KUKA KRL program: MyProgram_021().src

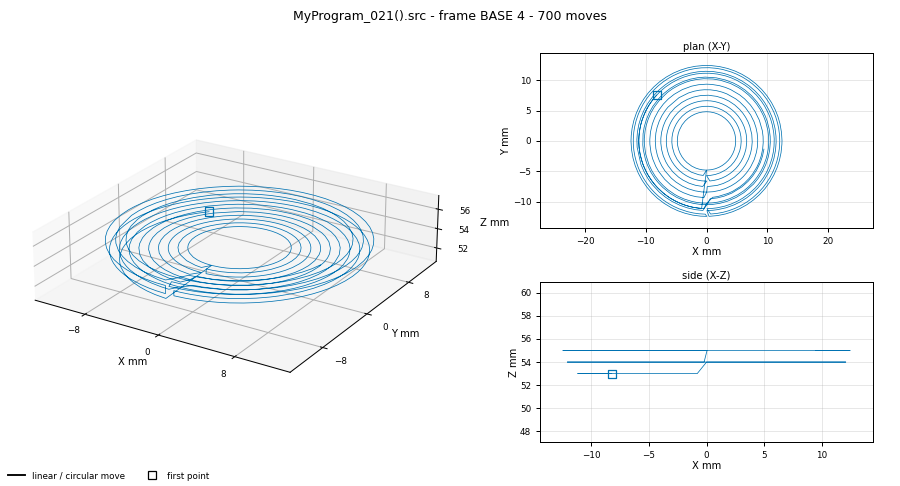
[picture p0: tool path of MyProgram_021().src in frame BASE 4, 700 of 700 moves have a stored position in this frame; points joined in program order, loops and branches not executed]
&ACCESS RVP
&REL 1
&PARAM TEMPLATE = C:\KRC\Roboter\Template\vorgabe
&PARAM EDITMASK = *
DEF MyProgram_021()
; ---- Setting reference (Base) ----
$BASE = BASE_DATA[4]

; --------------------------
; ---- Setting tool (TCP) ----
$TOOL = TOOL_DATA[3]
; --------------------------

$VEL.CP = VEL_APROX_PRINT
Startdeposition()
$VEL.CP = VEL_PRINT
LIN {X -8.217,Y 7.5391,Z 53,A 131.0651,B 24.783,C -3.3954,E1 24.879,E2 -48.9151} C_DIS
LIN {X -8.9524,Y 6.6493,Z 53,A 136.9358,B 24.785,C -3.3802,E1 24.8689,E2 -54.777} C_DIS
LIN {X -9.569,Y 5.7257,Z 53,A 142.7513,B 24.787,C -3.3647,E1 24.8603,E2 -60.5851} C_DIS
LIN {X -10.0751,Y 4.778,Z 53,A 148.3652,B 24.789,C -3.349,E1 24.8533,E2 -66.1916} C_DIS
LIN {X -10.6035,Y 3.4435,Z 53,A 154.2038,B 24.7919,C -3.3262,E1 24.8476,E2 -72.0082} C_DIS
LIN {X -10.8532,Y 2.565,Z 53,A 160.4775,B 24.7935,C -3.3127,E1 24.8431,E2 -78.2862} C_DIS
LIN {X -11.0746,Y 1.2842,Z 53,A 166.7328,B 24.7961,C -3.2919,E1 24.8405,E2 -84.5288} C_DIS
LIN {X -11.1513,Y 0.0898,Z 53,A 172.9449,B 24.7985,C -3.2728,E1 24.8398,E2 -90.7325} C_DIS
LIN {X -11.109,Y -0.9807,Z 53,A 178.5916,B 24.8006,C -3.2559,E1 24.8408,E2 -96.3727} C_DIS
LIN {X -10.9799,Y -1.9503,Z 53,A -176.0526,B 24.8024,C -3.2409,E1 24.8431,E2 -101.7244} C_DIS
LIN {X -10.6594,Y -3.2683,Z 53,A -170.537,B 24.8051,C -3.2194,E1 24.8469,E2 -107.2207} C_DIS
LIN {X -10.3597,Y -4.1289,Z 53,A -164.2287,B 24.8065,C -3.2074,E1 24.853,E2 -113.5357} C_DIS
LIN {X -9.7793,Y -5.3548,Z 53,A -158.8351,B 24.809,C -3.1872,E1 24.8596,E2 -118.9101} C_DIS
LIN {X -9.3116,Y -6.137,Z 53,A -152.506,B 24.8102,C -3.1773,E1 24.8689,E2 -125.2477} C_DIS
LIN {X -8.634,Y -7.0586,Z 53,A -146.9528,B 24.8118,C -3.1632,E1 24.8784,E2 -130.7935} C_DIS
LIN {X -7.9686,Y -7.8008,Z 53,A -141.4565,B 24.8131,C -3.1531,E1 24.889,E2 -136.2895} C_DIS
LIN {X -6.9974,Y -8.6837,Z 53,A -134.9618,B 24.8146,C -3.1401,E1 24.9027,E2 -142.7784} C_DIS
LIN {X -6.0499,Y -9.3683,Z 53,A -129.1842,B 24.8158,C -3.1301,E1 24.9159,E2 -148.5518} C_DIS
LIN {X -5.1971,Y -9.8667,Z 53,A -123.783,B 24.8165,C -3.1243,E1 24.9291,E2 -153.9546} C_DIS
LIN {X -4.1117,Y -10.3666,Z 53,A -117.7422,B 24.8172,C -3.1177,E1 24.9446,E2 -159.9938} C_DIS
LIN {X -3.1253,Y -10.7051,Z 53,A -112.1923,B 24.8176,C -3.1144,E1 24.9594,E2 -165.5458} C_DIS
LIN {X -2.0829,Y -10.9558,Z 53,A -106.4158,B 24.8178,C -3.113,E1 24.9752,E2 -171.3258} C_DIS
LIN {X -0.805,Y -11.1216,Z 53,A -100.2726,B 24.8181,C -3.1107,E1 24.9922,E2 -177.4669} C_DIS
LIN {X -0.805,Y -11.1216,Z 53,A -100.2726,B 24.8181,C -3.1107,E1 24.9922,E2 -177.4669} C_DIS
Enddeposition()
LIN {X 0.0024,Y -4.8102,Z 54,A -2.8466,B 0,C 0,E1 0.1598,E2 -269.9283} C_DIS
Startdeposition()
$VEL.CP = VEL_PRINT
LIN {X 0.8114,Y -4.7379,Z 54,A -2.8139,B 0,C 0,E1 0.1598,E2 -269.9282} C_DIS
LIN {X 1.4429,Y -4.5849,Z 54,A -2.7842,B 0,C 0,E1 0.1598,E2 -269.9282} C_DIS
LIN {X 2.0479,Y -4.3478,Z 54,A -2.7518,B 0,C 0,E1 0.1598,E2 -269.9282} C_DIS
LIN {X 2.6157,Y -4.0318,Z 54,A -2.7175,B 0,C 0,E1 0.1598,E2 -269.9281} C_DIS
LIN {X 3.1341,Y -3.6406,Z 54,A -2.6817,B 0,C 0,E1 0.1598,E2 -269.9281} C_DIS
LIN {X 3.5986,Y -3.1861,Z 54,A -2.6452,B 0,C 0,E1 0.1598,E2 -269.9281} C_DIS
LIN {X 3.9948,Y -2.6709,Z 54,A -2.6087,B 0,C 0,E1 0.1598,E2 -269.9281} C_DIS
LIN {X 4.319,Y -2.1081,Z 54,A -2.5727,B 0,C 0,E1 0.1598,E2 -269.9281} C_DIS
LIN {X 4.5648,Y -1.5065,Z 54,A -2.5379,B 0,C 0,E1 0.1598,E2 -269.9281} C_DIS
LIN {X 4.7263,Y -0.877,Z 54,A -2.5051,B 0,C 0,E1 0.1598,E2 -269.928} C_DIS
LIN {X 4.8021,Y -0.2316,Z 54,A -2.4748,B 0,C 0,E1 0.1598,E2 -269.928} C_DIS
LIN {X 4.7897,Y 0.4181,Z 54,A -2.4475,B 0,C 0,E1 0.1598,E2 -269.928} C_DIS
LIN {X 4.689,Y 1.0602,Z 54,A -2.4238,B 0,C 0,E1 0.1598,E2 -269.928} C_DIS
LIN {X 4.5023,Y 1.6826,Z 54,A -2.4041,B 0,C 0,E1 0.1598,E2 -269.9279} C_DIS
LIN {X 4.2321,Y 2.2734,Z 54,A -2.3889,B 0,C 0,E1 0.1598,E2 -269.9279} C_DIS
LIN {X 3.8894,Y 2.8255,Z 54,A -2.378,B 0,C 0,E1 0.1598,E2 -269.9278} C_DIS
LIN {X 3.4717,Y 3.3236,Z 54,A -2.3722,B 0,C 0,E1 0.1598,E2 -269.9278} C_DIS
LIN {X 2.9925,Y 3.7625,Z 54,A -2.3712,B 0,C 0,E1 0.1598,E2 -269.9278} C_DIS
LIN {X 2.4574,Y 4.1311,Z 54,A -2.3752,B 0,C 0,E1 0.1598,E2 -269.9277} C_DIS
LIN {X 1.8772,Y 4.4237,Z 54,A -2.3842,B 0,C 0,E1 0.1598,E2 -269.9277} C_DIS
LIN {X 1.263,Y 4.6358,Z 54,A -2.3978,B 0,C 0,E1 0.1598,E2 -269.9277} C_DIS
LIN {X 0.6263,Y 4.7649,Z 54,A -2.4158,B 0,C 0,E1 0.1598,E2 -269.9277} C_DIS
LIN {X -0.0221,Y 4.806,Z 54,A -2.4379,B 0,C 0,E1 0.1598,E2 -269.9277} C_DIS
LIN {X -0.6701,Y 4.7592,Z 54,A -2.4638,B 0,C 0,E1 0.1598,E2 -269.9277} C_DIS
LIN {X -1.3058,Y 4.6251,Z 54,A -2.4929,B 0,C 0,E1 0.1598,E2 -269.9277} C_DIS
LIN {X -1.9176,Y 4.4064,Z 54,A -2.5248,B 0,C 0,E1 0.1598,E2 -269.9278} C_DIS
LIN {X -2.4945,Y 4.1076,Z 54,A -2.5587,B 0,C 0,E1 0.1598,E2 -269.9278} C_DIS
LIN {X -3.0262,Y 3.734,Z 54,A -2.5941,B 0,C 0,E1 0.1598,E2 -269.928} C_DIS
LIN {X -3.5023,Y 3.2919,Z 54,A -2.6304,B 0,C 0,E1 0.1598,E2 -269.928} C_DIS
LIN {X -4.0104,Y 2.6581,Z 54,A -2.6759,B 0,C 0,E1 0.1598,E2 -269.9282} C_DIS
LIN {X -4.4662,Y 1.7787,Z 54,A -2.7298,B 0,C 0,E1 0.1598,E2 -269.9285} C_DIS
LIN {X -4.6661,Y 1.1608,Z 54,A -2.7636,B 0,C 0,E1 0.1598,E2 -269.9283} C_DIS
LIN {X -4.7799,Y 0.5214,Z 54,A -2.7949,B 0,C 0,E1 0.1598,E2 -269.9283} C_DIS
LIN {X -4.8062,Y -0.1275,Z 54,A -2.8234,B 0,C 0,E1 0.1598,E2 -269.9284} C_DIS
LIN {X -4.7448,Y -0.7741,Z 54,A -2.8486,B 0,C 0,E1 0.1598,E2 -269.9284} C_DIS
LIN {X -4.5964,Y -1.4062,Z 54,A -2.87,B 0,C 0,E1 0.1598,E2 -269.9284} C_DIS
LIN {X -4.3649,Y -2.013,Z 54,A -2.8873,B 0,C 0,E1 0.1598,E2 -269.9284} C_DIS
LIN {X -4.0539,Y -2.5829,Z 54,A -2.9001,B 0,C 0,E1 0.1598,E2 -269.9284} C_DIS
LIN {X -3.6667,Y -3.1042,Z 54,A -2.908,B 0,C 0,E1 0.1598,E2 -269.9284} C_DIS
LIN {X -3.2148,Y -3.57,Z 54,A -2.9113,B 0,C 0,E1 0.1598,E2 -269.9284} C_DIS
LIN {X -2.4084,Y -4.1653,Z 54,A -2.9069,B 0,C 0,E1 0.1598,E2 -269.9284} C_DIS
LIN {X -1.7765,Y -4.4675,Z 54,A -2.8967,B 0,C 0,E1 0.1598,E2 -269.9284} C_DIS
LIN {X -1.2443,Y -4.6427,Z 54,A -2.8847,B 0,C 0,E1 0.1598,E2 -269.9283} C_DIS
LIN {X -0.6958,Y -4.7564,Z 54,A -2.8694,B 0,C 0,E1 0.1598,E2 -269.9283} C_DIS
LIN {X 0.0024,Y -4.8102,Z 54,A -2.8461,B 0,C 0,E1 0.1598,E2 -269.9283} C_DIS
Enddeposition()
LIN {X 0.0024,Y -4.8102,Z 54,A -2.8461,B 0,C 0,E1 0.1598,E2 -269.9283} C_DIS
Startdeposition()
$VEL.CP = VEL_PRINT
LIN {X -0.5401,Y -5.685,Z 54,A -2.9028,B 0,C 0,E1 0.1598,E2 -269.9288} C_DIS
LIN {X -1.2716,Y -5.5684,Z 54,A -2.9252,B 0,C 0,E1 0.1598,E2 -269.9284} C_DIS
LIN {X -2.4971,Y -5.1425,Z 54,A -2.9519,B 0,C 0,E1 0.1598,E2 -269.9285} C_DIS
LIN {X -3.6673,Y -4.3804,Z 54,A -2.9623,B 0,C 0,E1 0.1598,E2 -269.9287} C_DIS
LIN {X -4.2148,Y -3.8632,Z 54,A -2.9605,B 0,C 0,E1 0.1598,E2 -269.9287} C_DIS
LIN {X -4.8402,Y -3.0421,Z 54,A -2.9484,B 0,C 0,E1 0.1598,E2 -269.9287} C_DIS
LIN {X -5.2993,Y -2.1427,Z 54,A -2.9267,B 0,C 0,E1 0.1598,E2 -269.9291} C_DIS
LIN {X -5.6197,Y -1.0212,Z 54,A -2.8909,B 0,C 0,E1 0.1598,E2 -269.929} C_DIS
LIN {X -5.7054,Y -0.2319,Z 54,A -2.8609,B 0,C 0,E1 0.1598,E2 -269.9286} C_DIS
LIN {X -5.6822,Y 0.5616,Z 54,A -2.8264,B 0,C 0,E1 0.1598,E2 -269.9286} C_DIS
LIN {X -5.5516,Y 1.3448,Z 54,A -2.7884,B 0,C 0,E1 0.1598,E2 -269.9285} C_DIS
LIN {X -5.3117,Y 2.1019,Z 54,A -2.7474,B 0,C 0,E1 0.1598,E2 -269.9284} C_DIS
LIN {X -4.9675,Y 2.8175,Z 54,A -2.7044,B 0,C 0,E1 0.1598,E2 -269.9284} C_DIS
LIN {X -4.5288,Y 3.4791,Z 54,A -2.6603,B 0,C 0,E1 0.1598,E2 -269.9282} C_DIS
LIN {X -4.0028,Y 4.0739,Z 54,A -2.6157,B 0,C 0,E1 0.1598,E2 -269.9281} C_DIS
LIN {X -3.3989,Y 4.5894,Z 54,A -2.5716,B 0,C 0,E1 0.1598,E2 -269.928} C_DIS
LIN {X -2.7293,Y 5.016,Z 54,A -2.5289,B 0,C 0,E1 0.1598,E2 -269.9279} C_DIS
LIN {X -2.0072,Y 5.3461,Z 54,A -2.4883,B 0,C 0,E1 0.1598,E2 -269.9278} C_DIS
LIN {X -1.2463,Y 5.5726,Z 54,A -2.4506,B 0,C 0,E1 0.1598,E2 -269.9278} C_DIS
LIN {X -0.4613,Y 5.6909,Z 54,A -2.4167,B 0,C 0,E1 0.1598,E2 -269.9277} C_DIS
LIN {X 0.3324,Y 5.7012,Z 54,A -2.387,B 0,C 0,E1 0.1598,E2 -269.9277} C_DIS
LIN {X 1.1202,Y 5.6008,Z 54,A -2.3622,B 0,C 0,E1 0.1598,E2 -269.9276} C_DIS
LIN {X 1.8858,Y 5.3907,Z 54,A -2.3429,B 0,C 0,E1 0.1598,E2 -269.9276} C_DIS
LIN {X 2.6148,Y 5.0763,Z 54,A -2.3293,B 0,C 0,E1 0.1598,E2 -269.9276} C_DIS
LIN {X 3.294,Y 4.6652,Z 54,A -2.3218,B 0,C 0,E1 0.1598,E2 -269.9276} C_DIS
LIN {X 3.9093,Y 4.1634,Z 54,A -2.3204,B 0,C 0,E1 0.1598,E2 -269.9276} C_DIS
LIN {X 4.4488,Y 3.5808,Z 54,A -2.3253,B 0,C 0,E1 0.1598,E2 -269.9277} C_DIS
LIN {X 4.9028,Y 2.9295,Z 54,A -2.3363,B 0,C 0,E1 0.1598,E2 -269.9278} C_DIS
LIN {X 5.2613,Y 2.221,Z 54,A -2.3533,B 0,C 0,E1 0.1598,E2 -269.9278} C_DIS
LIN {X 5.5168,Y 1.4694,Z 54,A -2.3759,B 0,C 0,E1 0.1598,E2 -269.9279} C_DIS
LIN {X 5.669,Y 0.6903,Z 54,A -2.4036,B 0,C 0,E1 0.1598,E2 -269.9279} C_DIS
LIN {X 5.7096,Y -0.1026,Z 54,A -2.4359,B 0,C 0,E1 0.1598,E2 -269.928} C_DIS
LIN {X 5.6414,Y -0.8937,Z 54,A -2.4722,B 0,C 0,E1 0.1598,E2 -269.928} C_DIS
LIN {X 5.4629,Y -1.6674,Z 54,A -2.5118,B 0,C 0,E1 0.1598,E2 -269.9281} C_DIS
LIN {X 5.0471,Y -2.6857,Z 54,A -2.5704,B 0,C 0,E1 0.1598,E2 -269.9284} C_DIS
LIN {X 4.5814,Y -3.4121,Z 54,A -2.6188,B 0,C 0,E1 0.1598,E2 -269.9282} C_DIS
LIN {X 4.0192,Y -4.0668,Z 54,A -2.6674,B 0,C 0,E1 0.1598,E2 -269.9282} C_DIS
LIN {X 3.1947,Y -4.7411,Z 54,A -2.7265,B 0,C 0,E1 0.1598,E2 -269.9282} C_DIS
LIN {X 2.2685,Y -5.2416,Z 54,A -2.7819,B 0,C 0,E1 0.1598,E2 -269.9282} C_DIS
LIN {X 1.4728,Y -5.517,Z 54,A -2.823,B 0,C 0,E1 0.1598,E2 -269.9282} C_DIS
LIN {X 0.6457,Y -5.6742,Z 54,A -2.86,B 0,C 0,E1 0.1598,E2 -269.9282} C_DIS
LIN {X 0.015,Y -5.7133,Z 54,A -2.8848,B 0,C 0,E1 0.1598,E2 -269.9282} C_DIS
Enddeposition()
LIN {X 0.015,Y -5.7133,Z 54,A -2.8848,B 0,C 0,E1 0.1598,E2 -269.9282} C_DIS
Startdeposition()
$VEL.CP = VEL_PRINT
LIN {X 0.5509,Y -6.5971,Z 54,A -87.2231,B 10.8099,C -0.6837,E1 10.8502,E2 -187.2658} C_DIS
LIN {X 1.2406,Y -6.5027,Z 54,A -81.5321,B 10.8098,C -0.6867,E1 10.8658,E2 -192.9584} C_DIS
LIN {X 1.9167,Y -6.338,Z 54,A -75.4134,B 10.8094,C -0.6921,E1 10.8823,E2 -199.0813} C_DIS
LIN {X 2.5716,Y -6.1025,Z 54,A -69.4109,B 10.809,C -0.699,E1 10.898,E2 -205.0878} C_DIS
LIN {X 3.1981,Y -5.7991,Z 54,A -63.3454,B 10.8084,C -0.7077,E1 10.913,E2 -211.1579} C_DIS
LIN {X 3.7889,Y -5.431,Z 54,A -57.3881,B 10.8078,C -0.7176,E1 10.9269,E2 -217.1193} C_DIS
LIN {X 4.3378,Y -5.0031,Z 54,A -51.4315,B 10.807,C -0.729,E1 10.9397,E2 -223.0801} C_DIS
LIN {X 4.8389,Y -4.52,Z 54,A -45.4727,B 10.8062,C -0.7415,E1 10.9514,E2 -229.0434} C_DIS
LIN {X 5.2864,Y -3.9869,Z 54,A -39.5211,B 10.8052,C -0.7552,E1 10.9617,E2 -234.9994} C_DIS
LIN {X 5.6755,Y -3.4099,Z 54,A -33.5711,B 10.8042,C -0.7698,E1 10.9707,E2 -240.9538} C_DIS
LIN {X 6.0017,Y -2.7951,Z 54,A -27.5272,B 10.8031,C -0.7856,E1 10.9782,E2 -247.0025} C_DIS
LIN {X 6.261,Y -2.1493,Z 54,A -21.7054,B 10.802,C -0.8012,E1 10.9838,E2 -252.8278} C_DIS
LIN {X 6.4923,Y -1.3106,Z 54,A -13.5868,B 10.8002,C -0.8245,E1 10.989,E2 -260.9553} C_DIS
LIN {X 6.6143,Y -0.3017,Z 54,A -5.704,B 10.7986,C -0.8461,E1 10.991,E2 -268.8389} C_DIS
LIN {X 6.6115,Y 0.3653,Z 54,A -0.049,B 10.7973,C -0.8621,E1 10.9906,E2 -274.497} C_DIS
LIN {X 6.5419,Y 1.0288,Z 54,A 5.6543,B 10.7961,C -0.8781,E1 10.9885,E2 -280.2032} C_DIS
LIN {X 6.4055,Y 1.6818,Z 54,A 11.4383,B 10.7948,C -0.8941,E1 10.9848,E2 -285.9903} C_DIS
LIN {X 6.2033,Y 2.3176,Z 54,A 17.1038,B 10.7935,C -0.9092,E1 10.9796,E2 -291.6578} C_DIS
LIN {X 5.9385,Y 2.9299,Z 54,A 22.7809,B 10.7923,C -0.9236,E1 10.9729,E2 -297.3367} C_DIS
LIN {X 5.6136,Y 3.5125,Z 54,A 28.5721,B 10.7911,C -0.9376,E1 10.9647,E2 -303.1298} C_DIS
LIN {X 5.2308,Y 4.0589,Z 54,A 34.0695,B 10.7901,C -0.9498,E1 10.9556,E2 -308.6272} C_DIS
LIN {X 4.7971,Y 4.5658,Z 54,A 39.8741,B 10.789,C -0.9619,E1 10.9447,E2 -314.4329} C_DIS
LIN {X 4.3134,Y 5.0254,Z 54,A 45.9575,B 10.788,C -0.9735,E1 10.9321,E2 -320.5183} C_DIS
LIN {X 3.7838,Y 5.4311,Z 54,A 51.0615,B 10.7873,C -0.9813,E1 10.9206,E2 -325.6192} C_DIS
LIN {X 3.2195,Y 5.7868,Z 54,A 57.0813,B 10.7865,C -0.99,E1 10.9062,E2 -331.6396} C_DIS
LIN {X 2.6205,Y 6.0802,Z 54,A 62.9866,B 10.7859,C -0.9968,E1 10.8912,E2 -337.5448} C_DIS
LIN {X 1.9954,Y 6.3135,Z 54,A 68.3454,B 10.7855,C -1.0012,E1 10.877,E2 -342.9003} C_DIS
LIN {X 1.3504,Y 6.4835,Z 54,A 74.382,B 10.7851,C -1.0051,E1 10.8606,E2 -348.9363} C_DIS
LIN {X 0.6911,Y 6.5857,Z 54,A 80.1461,B 10.7849,C -1.0069,E1 10.8447,E2 -354.6982} C_DIS
LIN {X 0.025,Y 6.6213,Z 54,A 86.1217,B 10.7849,C -1.0073,E1 10.828,E2 -360.6722} C_DIS
LIN {X -0.6412,Y 6.588,Z 54,A 91.4727,B 10.7851,C -1.0055,E1 10.8131,E2 -366.0184} C_DIS
LIN {X -1.3012,Y 6.4913,Z 54,A 97.5304,B 10.7853,C -1.0026,E1 10.7965,E2 -372.074} C_DIS
LIN {X -1.9473,Y 6.3258,Z 54,A 103.3049,B 10.7858,C -0.9978,E1 10.781,E2 -377.845} C_DIS
LIN {X -2.5738,Y 6.0973,Z 54,A 108.6956,B 10.7863,C -0.9917,E1 10.767,E2 -383.2303} C_DIS
LIN {X -3.1758,Y 5.8099,Z 54,A 114.887,B 10.7871,C -0.9837,E1 10.7516,E2 -389.4193} C_DIS
LIN {X -3.7448,Y 5.4616,Z 54,A 120.7148,B 10.7879,C -0.9744,E1 10.738,E2 -395.2431} C_DIS
LIN {X -4.2752,Y 5.0568,Z 54,A 126.5487,B 10.7888,C -0.9638,E1 10.7253,E2 -401.0728} C_DIS
LIN {X -4.7621,Y 4.6009,Z 54,A 132.3688,B 10.7899,C -0.952,E1 10.7137,E2 -406.8886} C_DIS
LIN {X -5.2006,Y 4.0982,Z 54,A 138.2296,B 10.791,C -0.939,E1 10.7033,E2 -412.7452} C_DIS
LIN {X -5.5864,Y 3.554,Z 54,A 144.0551,B 10.7922,C -0.9251,E1 10.6942,E2 -418.5663} C_DIS
LIN {X -5.9156,Y 2.9739,Z 54,A 149.8973,B 10.7934,C -0.9102,E1 10.6865,E2 -424.4044} C_DIS
LIN {X -6.185,Y 2.3637,Z 54,A 156.0252,B 10.7947,C -0.8942,E1 10.6801,E2 -430.5292} C_DIS
LIN {X -6.3885,Y 1.7285,Z 54,A 161.4712,B 10.796,C -0.8789,E1 10.6758,E2 -435.9697} C_DIS
LIN {X -6.5322,Y 1.0771,Z 54,A 167.4911,B 10.7973,C -0.8622,E1 10.6726,E2 -441.9864} C_DIS
LIN {X -6.6065,Y 0.4143,Z 54,A 173.2032,B 10.7986,C -0.8459,E1 10.6712,E2 -447.6943} C_DIS
LIN {X -6.6166,Y -0.2527,Z 54,A 179.2499,B 10.7999,C -0.8289,E1 10.6714,E2 -453.7385} C_DIS
LIN {X -6.5573,Y -0.9171,Z 54,A -174.9302,B 10.8011,C -0.8125,E1 10.6733,E2 -459.5552} C_DIS
LIN {X -6.4319,Y -1.5722,Z 54,A -169.0783,B 10.8023,C -0.7964,E1 10.6767,E2 -465.4045} C_DIS
LIN {X -6.2413,Y -2.2114,Z 54,A -163.2119,B 10.8034,C -0.7807,E1 10.6818,E2 -471.2685} C_DIS
LIN {X -5.9868,Y -2.828,Z 54,A -157.097,B 10.8045,C -0.7653,E1 10.6887,E2 -477.3828} C_DIS
LIN {X -5.6708,Y -3.4155,Z 54,A -151.7315,B 10.8055,C -0.7519,E1 10.6962,E2 -482.7444} C_DIS
LIN {X -5.2993,Y -3.9695,Z 54,A -145.6359,B 10.8064,C -0.7384,E1 10.706,E2 -488.8401} C_DIS
LIN {X -4.873,Y -4.4824,Z 54,A -139.8003,B 10.8072,C -0.7264,E1 10.7167,E2 -494.675} C_DIS
LIN {X -4.3971,Y -4.9498,Z 54,A -133.9626,B 10.8079,C -0.7156,E1 10.7286,E2 -500.5125} C_DIS
LIN {X -3.876,Y -5.366,Z 54,A -128.0686,B 10.8085,C -0.7061,E1 10.7417,E2 -506.407} C_DIS
LIN {X -3.3166,Y -5.7294,Z 54,A -122.302,B 10.809,C -0.6981,E1 10.7555,E2 -512.174} C_DIS
LIN {X -2.7232,Y -6.034,Z 54,A -116.6793,B 10.8094,C -0.6916,E1 10.7696,E2 -517.7967} C_DIS
LIN {X -2.1026,Y -6.2783,Z 54,A -110.7462,B 10.8098,C -0.6866,E1 10.7852,E2 -523.7319} C_DIS
LIN {X -1.4603,Y -6.4582,Z 54,A -104.7879,B 10.81,C -0.6834,E1 10.8013,E2 -529.6929} C_DIS
LIN {X -0.8028,Y -6.5706,Z 54,A -99.091,B 10.81,C -0.6817,E1 10.8171,E2 -535.3916} C_DIS
LIN {X 0.0293,Y -6.6199,Z 54,A -94.6585,B 10.8102,C -0.679,E1 10.8294,E2 -539.8122} C_DIS
Enddeposition()
LIN {X 0.0293,Y -6.6199,Z 54,A -94.6585,B 10.8102,C -0.679,E1 10.8294,E2 -539.8122} C_DIS
Startdeposition()
$VEL.CP = VEL_PRINT
LIN {X -0.6225,Y -7.5046,Z 54,A -102.6208,B 16.025,C -1.3921,E1 16.0632,E2 -532.9802} C_DIS
LIN {X -1.8167,Y -7.3038,Z 54,A -109.992,B 16.0245,C -1.398,E1 16.0431,E2 -525.6172} C_DIS
LIN {X -2.8776,Y -6.9579,Z 54,A -119.7083,B 16.0239,C -1.4043,E1 16.0175,E2 -515.8927} C_DIS
LIN {X -3.8717,Y -6.4538,Z 54,A -127.4228,B 16.023,C -1.4152,E1 15.9986,E2 -508.1826} C_DIS
LIN {X -4.5958,Y -5.9636,Z 54,A -134.6216,B 16.0221,C -1.4258,E1 15.9823,E2 -500.9818} C_DIS
LIN {X -5.5747,Y -5.0632,Z 54,A -145.3901,B 16.0203,C -1.4458,E1 15.961,E2 -490.213} C_DIS
LIN {X -6.3278,Y -4.0739,Z 54,A -152.413,B 16.0186,C -1.4655,E1 15.9494,E2 -483.207} C_DIS
LIN {X -6.6994,Y -3.4399,Z 54,A -160.3978,B 16.0171,C -1.4816,E1 15.9386,E2 -475.2132} C_DIS
LIN {X -7.1179,Y -2.4589,Z 54,A -168.4783,B 16.0152,C -1.5033,E1 15.9306,E2 -467.1385} C_DIS
LIN {X -7.3822,Y -1.4676,Z 54,A -175.4984,B 16.0132,C -1.5243,E1 15.926,E2 -460.1283} C_DIS
LIN {X -7.5214,Y -0.3734,Z 54,A 175.9813,B 16.011,C -1.5487,E1 15.9236,E2 -451.6145} C_DIS
LIN {X -7.5155,Y 0.4617,Z 54,A 169.1679,B 16.0091,C -1.5679,E1 15.9242,E2 -444.8049} C_DIS
LIN {X -7.3994,Y 1.4007,Z 54,A 161.3843,B 16.0071,C -1.5896,E1 15.9276,E2 -437.0258} C_DIS
LIN {X -7.113,Y 2.459,Z 54,A 153.6683,B 16.0048,C -1.6125,E1 15.9337,E2 -429.3211} C_DIS
LIN {X -6.7458,Y 3.3445,Z 54,A 146.0273,B 16.0028,C -1.6326,E1 15.9425,E2 -421.686} C_DIS
LIN {X -6.0298,Y 4.5097,Z 54,A 134.9592,B 16.0002,C -1.6592,E1 15.9595,E2 -410.6256} C_DIS
LIN {X -5.1947,Y 5.4498,Z 54,A 124.8201,B 15.998,C -1.6805,E1 15.9792,E2 -400.4935} C_DIS
LIN {X -4.0818,Y 6.3282,Z 54,A 114.6963,B 15.996,C -1.6996,E1 16.002,E2 -390.3826} C_DIS
LIN {X -3.1479,Y 6.8357,Z 54,A 106.9875,B 15.9948,C -1.7112,E1 16.0212,E2 -382.6825} C_DIS
LIN {X -2.1551,Y 7.2149,Z 54,A 98.4866,B 15.994,C -1.7194,E1 16.0436,E2 -374.1855} C_DIS
LIN {X -1.0372,Y 7.4539,Z 54,A 90.2017,B 15.9934,C -1.7254,E1 16.0663,E2 -365.9084} C_DIS
LIN {X 0.2973,Y 7.5246,Z 54,A 78.7875,B 15.9934,C -1.7252,E1 16.0981,E2 -354.4929} C_DIS
LIN {X 1.6715,Y 7.3371,Z 54,A 69.3006,B 15.9936,C -1.7231,E1 16.1242,E2 -345.015} C_DIS
LIN {X 2.8177,Y 6.9834,Z 54,A 60.6987,B 15.9943,C -1.7167,E1 16.1469,E2 -336.4172} C_DIS
LIN {X 3.6825,Y 6.5674,Z 54,A 52.9985,B 15.9953,C -1.7066,E1 16.166,E2 -328.7149} C_DIS
LIN {X 4.6404,Y 5.9293,Z 54,A 43.8028,B 15.9969,C -1.6913,E1 16.1869,E2 -319.5156} C_DIS
LIN {X 5.4921,Y 5.1453,Z 54,A 35.6502,B 15.9984,C -1.6764,E1 16.2033,E2 -311.3644} C_DIS
LIN {X 5.9993,Y 4.543,Z 54,A 29.3624,B 15.9999,C -1.662,E1 16.2142,E2 -305.0724} C_DIS
LIN {X 6.4398,Y 3.8903,Z 54,A 23.8542,B 16.0011,C -1.6496,E1 16.2225,E2 -299.5641} C_DIS
LIN {X 6.813,Y 3.197,Z 54,A 17.6229,B 16.0028,C -1.6333,E1 16.2303,E2 -293.3276} C_DIS
LIN {X 7.1086,Y 2.4672,Z 54,A 11.9864,B 16.0042,C -1.6187,E1 16.2359,E2 -287.6893} C_DIS
LIN {X 7.451,Y 1.0886,Z 54,A -0.0547,B 16.0077,C -1.5827,E1 16.2427,E2 -275.6318} C_DIS
LIN {X 7.5274,Y -0.1798,Z 54,A -8.7198,B 16.01,C -1.5589,E1 16.2433,E2 -266.9643} C_DIS
LIN {X 7.4365,Y -1.1791,Z 54,A -16.2028,B 16.012,C -1.5373,E1 16.2408,E2 -259.4749} C_DIS
LIN {X 7.233,Y -2.097,Z 54,A -23.6408,B 16.0141,C -1.5155,E1 16.2356,E2 -252.0278} C_DIS
LIN {X 6.8961,Y -3.023,Z 54,A -31.0943,B 16.0159,C -1.495,E1 16.2279,E2 -244.5669} C_DIS
LIN {X 6.4181,Y -3.9328,Z 54,A -38.3227,B 16.0176,C -1.477,E1 16.218,E2 -237.3344} C_DIS
LIN {X 5.9631,Y -4.5964,Z 54,A -44.8089,B 16.019,C -1.4605,E1 16.2073,E2 -230.8395} C_DIS
LIN {X 5.4213,Y -5.2248,Z 54,A -51.1979,B 16.0203,C -1.446,E1 16.1952,E2 -224.4438} C_DIS
LIN {X 4.5718,Y -5.9821,Z 54,A -59.6646,B 16.0218,C -1.4295,E1 16.177,E2 -215.97} C_DIS
LIN {X 3.6739,Y -6.5678,Z 54,A -67.1039,B 16.0227,C -1.4182,E1 16.1593,E2 -208.5282} C_DIS
LIN {X 2.7544,Y -7.0092,Z 54,A -76.2961,B 16.024,C -1.4039,E1 16.1358,E2 -199.3206} C_DIS
LIN {X 1.7894,Y -7.3144,Z 54,A -84.2551,B 16.0246,C -1.3964,E1 16.1143,E2 -191.3546} C_DIS
LIN {X 0.1158,Y -7.5288,Z 54,A -95.2263,B 16.0248,C -1.3945,E1 16.0838,E2 -180.3877} C_DIS
LIN {X 0.1158,Y -7.5288,Z 54,A -95.2263,B 16.0248,C -1.3945,E1 16.0838,E2 -180.3877} C_DIS
Enddeposition()
LIN {X 0.0276,Y -8.431,Z 54,A -95.6356,B 21.2021,C -2.3401,E1 21.3276,E2 -181.2403} C_DIS
Startdeposition()
$VEL.CP = VEL_PRINT
LIN {X 1.1282,Y -8.3607,Z 54,A -86.6538,B 21.2013,C -2.3478,E1 21.3526,E2 -190.237} C_DIS
LIN {X 2.1816,Y -8.1461,Z 54,A -80.552,B 21.201,C -2.3503,E1 21.3692,E2 -196.3356} C_DIS
LIN {X 3.1517,Y -7.8259,Z 54,A -72.727,B 21.1998,C -2.3618,E1 21.3897,E2 -204.1731} C_DIS
LIN {X 4.0868,Y -7.3743,Z 54,A -66.1117,B 21.1988,C -2.3711,E1 21.4062,E2 -210.7922} C_DIS
LIN {X 4.793,Y -6.9366,Z 54,A -60.5207,B 21.1977,C -2.3811,E1 21.4192,E2 -216.3889} C_DIS
LIN {X 5.4529,Y -6.4319,Z 54,A -55.0288,B 21.1965,C -2.392,E1 21.4312,E2 -221.8859} C_DIS
LIN {X 6.0604,Y -5.865,Z 54,A -49.224,B 21.1951,C -2.4054,E1 21.4428,E2 -227.6986} C_DIS
LIN {X 6.6073,Y -5.2395,Z 54,A -43.6532,B 21.1936,C -2.4189,E1 21.4527,E2 -233.2759} C_DIS
LIN {X 7.2505,Y -4.3132,Z 54,A -35.7516,B 21.1913,C -2.4402,E1 21.4647,E2 -241.189} C_DIS
LIN {X 7.8487,Y -3.0961,Z 54,A -26.2647,B 21.1883,C -2.4677,E1 21.4756,E2 -250.6899} C_DIS
LIN {X 8.2114,Y -1.9171,Z 54,A -18.4973,B 21.1858,C -2.4893,E1 21.4814,E2 -258.4634} C_DIS
LIN {X 8.3703,Y -1.0261,Z 54,A -12.4611,B 21.1838,C -2.5072,E1 21.4839,E2 -264.5064} C_DIS
LIN {X 8.434,Y 0.1704,Z 54,A -4.3489,B 21.1811,C -2.5315,E1 21.4845,E2 -272.6281} C_DIS
LIN {X 8.3439,Y 1.2438,Z 54,A 3.097,B 21.1785,C -2.554,E1 21.4822,E2 -280.0833} C_DIS
LIN {X 8.1431,Y 2.2032,Z 54,A 9.6166,B 21.1763,C -2.5726,E1 21.478,E2 -286.6089} C_DIS
LIN {X 7.8382,Y 3.1191,Z 54,A 16.8641,B 21.1738,C -2.5943,E1 21.4709,E2 -293.8678} C_DIS
LIN {X 7.284,Y 4.2492,Z 54,A 24.373,B 21.1718,C -2.6112,E1 21.4611,E2 -301.3762} C_DIS
LIN {X 6.4171,Y 5.4748,Z 54,A 35.8226,B 21.1684,C -2.6404,E1 21.4417,E2 -312.8412} C_DIS
LIN {X 5.4929,Y 6.3959,Z 54,A 43.1332,B 21.1671,C -2.651,E1 21.4269,E2 -320.1452} C_DIS
LIN {X 4.8107,Y 6.929,Z 54,A 50.8409,B 21.1651,C -2.6678,E1 21.4094,E2 -327.867} C_DIS
LIN {X 3.3598,Y 7.7376,Z 54,A 60.6789,B 21.1641,C -2.6763,E1 21.3849,E2 -337.6964} C_DIS
LIN {X 2.5856,Y 8.0297,Z 54,A 66.6613,B 21.1634,C -2.6821,E1 21.3691,E2 -343.6807} C_DIS
LIN {X 1.6802,Y 8.2667,Z 54,A 72.7242,B 21.1631,C -2.6846,E1 21.3526,E2 -349.7404} C_DIS
LIN {X 0.6449,Y 8.4114,Z 54,A 79.6912,B 21.163,C -2.6855,E1 21.3333,E2 -356.7041} C_DIS
LIN {X -0.3753,Y 8.4245,Z 54,A 86.5907,B 21.1631,C -2.6842,E1 21.3141,E2 -363.6} C_DIS
LIN {X -1.1879,Y 8.3476,Z 54,A 92.1541,B 21.1635,C -2.6814,E1 21.2986,E2 -369.1601} C_DIS
LIN {X -1.9893,Y 8.1933,Z 54,A 97.5698,B 21.164,C -2.6768,E1 21.2839,E2 -374.571} C_DIS
LIN {X -2.9656,Y 7.8971,Z 54,A 106.1126,B 21.1647,C -2.6708,E1 21.2614,E2 -383.1169} C_DIS
LIN {X -4.5341,Y 7.114,Z 54,A 119.2976,B 21.167,C -2.6522,E1 21.2296,E2 -396.2969} C_DIS
LIN {X -6.3433,Y 5.561,Z 54,A 132.236,B 21.1712,C -2.6163,E1 21.2033,E2 -409.1985} C_DIS
LIN {X -6.797,Y 4.9972,Z 54,A 138.1223,B 21.1727,C -2.6039,E1 21.1933,E2 -415.0838} C_DIS
LIN {X -7.3259,Y 4.1838,Z 54,A 145.1701,B 21.1748,C -2.5862,E1 21.1831,E2 -422.1255} C_DIS
LIN {X -7.7974,Y 3.2156,Z 54,A 151.5342,B 21.1771,C -2.5661,E1 21.1758,E2 -428.4753} C_DIS
LIN {X -8.1419,Y 2.2076,Z 54,A 159.4933,B 21.1796,C -2.5445,E1 21.1691,E2 -436.4289} C_DIS
LIN {X -8.3386,Y 1.2767,Z 54,A 166.1394,B 21.1818,C -2.5251,E1 21.1658,E2 -443.0678} C_DIS
LIN {X -8.437,Y 0.0383,Z 54,A 175.2854,B 21.1847,C -2.4991,E1 21.1648,E2 -452.2073} C_DIS
LIN {X -8.3426,Y -1.2521,Z 54,A -176.4078,B 21.1876,C -2.4733,E1 21.1673,E2 -460.5015} C_DIS
LIN {X -8.087,Y -2.4023,Z 54,A -168.478,B 21.1902,C -2.4503,E1 21.1728,E2 -468.4226} C_DIS
LIN {X -7.7669,Y -3.2808,Z 54,A -162.6573,B 21.1921,C -2.4332,E1 21.1787,E2 -474.2346} C_DIS
LIN {X -7.3595,Y -4.1226,Z 54,A -155.721,B 21.1939,C -2.4165,E1 21.1876,E2 -481.1688} C_DIS
LIN {X -6.848,Y -4.9279,Z 54,A -148.0345,B 21.1956,C -2.4012,E1 21.1999,E2 -488.8579} C_DIS
LIN {X -5.7863,Y -6.1377,Z 54,A -138.2423,B 21.198,C -2.3783,E1 21.2186,E2 -498.6373} C_DIS
LIN {X -5.0175,Y -6.7826,Z 54,A -131.5962,B 21.1993,C -2.3664,E1 21.2332,E2 -505.2798} C_DIS
LIN {X -3.9696,Y -7.4436,Z 54,A -121.7245,B 21.2003,C -2.3566,E1 21.257,E2 -515.1595} C_DIS
LIN {X -3.0466,Y -7.8673,Z 54,A -115.5849,B 21.2011,C -2.3489,E1 21.2729,E2 -521.2941} C_DIS
LIN {X -1.8873,Y -8.2177,Z 54,A -108.0527,B 21.2018,C -2.3428,E1 21.2931,E2 -528.823} C_DIS
LIN {X -0.8347,Y -8.3951,Z 54,A -100.2493,B 21.2018,C -2.3424,E1 21.3147,E2 -536.6324} C_DIS
LIN {X 0.0276,Y -8.431,Z 54,A -96.3606,B 21.2023,C -2.3382,E1 21.3255,E2 -540.5102} C_DIS
Enddeposition()
LIN {X 0.0276,Y -8.431,Z 54,A -96.3606,B 21.2023,C -2.3382,E1 21.3255,E2 -540.5102} C_DIS
Startdeposition()
$VEL.CP = VEL_PRINT
LIN {X -0.4267,Y -9.3338,Z 54,A -101.7866,B 24.8148,C -3.1386,E1 24.9882,E2 -536.0191} C_DIS
LIN {X -1.7131,Y -9.1852,Z 54,A -109.633,B 24.8145,C -3.1406,E1 24.9665,E2 -528.1711} C_DIS
LIN {X -2.6403,Y -8.9621,Z 54,A -115.8561,B 24.8142,C -3.1433,E1 24.9498,E2 -521.9447} C_DIS
LIN {X -3.7967,Y -8.5324,Z 54,A -121.3225,B 24.8129,C -3.1546,E1 24.9356,E2 -516.4936} C_DIS
LIN {X -4.5899,Y -8.1367,Z 54,A -129.6831,B 24.8127,C -3.1564,E1 24.9149,E2 -508.1141} C_DIS
LIN {X -5.8923,Y -7.2514,Z 54,A -138.7667,B 24.8106,C -3.1732,E1 24.8946,E2 -499.0384} C_DIS
LIN {X -6.8805,Y -6.3198,Z 54,A -147.8405,B 24.8086,C -3.1898,E1 24.8769,E2 -489.9655} C_DIS
LIN {X -7.856,Y -5.0569,Z 54,A -155.6466,B 24.8057,C -3.2142,E1 24.8642,E2 -482.1798} C_DIS
LIN {X -8.3477,Y -4.1947,Z 54,A -163.2323,B 24.8038,C -3.2298,E1 24.8542,E2 -474.5912} C_DIS
LIN {X -8.8563,Y -2.9775,Z 54,A -170.2475,B 24.801,C -3.2526,E1 24.8472,E2 -467.5914} C_DIS
LIN {X -9.1423,Y -1.92,Z 54,A -178.3476,B 24.7985,C -3.2726,E1 24.842,E2 -459.4918} C_DIS
LIN {X -9.3241,Y -0.5379,Z 54,A 174.2677,B 24.7953,C -3.2987,E1 24.8399,E2 -452.1252} C_DIS
LIN {X -9.3366,Y 0.2473,Z 54,A 169.4988,B 24.7934,C -3.3136,E1 24.8399,E2 -447.3634} C_DIS
LIN {X -9.224,Y 1.4786,Z 54,A 161.5798,B 24.7905,C -3.3371,E1 24.8425,E2 -439.4534} C_DIS
LIN {X -8.9122,Y 2.7996,Z 54,A 153.0447,B 24.7873,C -3.3625,E1 24.8485,E2 -430.9295} C_DIS
LIN {X -8.5158,Y 3.8321,Z 54,A 146.6818,B 24.7847,C -3.3825,E1 24.8552,E2 -424.5792} C_DIS
LIN {X -7.8959,Y 4.9926,Z 54,A 137.6553,B 24.7818,C -3.4048,E1 24.8677,E2 -415.559} C_DIS
LIN {X -7.1061,Y 6.0634,Z 54,A 129.4411,B 24.7792,C -3.4255,E1 24.8819,E2 -407.356} C_DIS
LIN {X -6.2611,Y 6.9355,Z 54,A 122.1458,B 24.7769,C -3.4426,E1 24.8965,E2 -400.0714} C_DIS
LIN {X -5.3216,Y 7.6774,Z 54,A 114.7177,B 24.775,C -3.4573,E1 24.9131,E2 -392.652} C_DIS
LIN {X -3.968,Y 8.4577,Z 54,A 103.426,B 24.7733,C -3.4704,E1 24.9411,E2 -381.3609} C_DIS
LIN {X -2.4474,Y 9.0159,Z 54,A 94.7461,B 24.7716,C -3.4836,E1 24.9641,E2 -372.6972} C_DIS
LIN {X -1.3109,Y 9.2509,Z 54,A 87.9433,B 24.7708,C -3.4893,E1 24.9828,E2 -365.9015} C_DIS
LIN {X -0.0062,Y 9.3434,Z 54,A 80.5908,B 24.7702,C -3.4936,E1 25.0033,E2 -358.5577} C_DIS
LIN {X 0.8706,Y 9.3027,Z 54,A 74.0291,B 24.7707,C -3.4899,E1 25.0216,E2 -351.9905} C_DIS
LIN {X 2.1604,Y 9.0902,Z 54,A 65.9239,B 24.7712,C -3.4861,E1 25.0437,E2 -343.8863} C_DIS
LIN {X 3.11,Y 8.8095,Z 54,A 60.4635,B 24.7716,C -3.4835,E1 25.0582,E2 -338.4303} C_DIS
LIN {X 3.975,Y 8.4544,Z 54,A 54.4012,B 24.7726,C -3.4759,E1 25.0736,E2 -332.3651} C_DIS
LIN {X 5.4357,Y 7.5985,Z 54,A 44.6319,B 24.7742,C -3.4632,E1 25.0967,E2 -322.5969} C_DIS
LIN {X 6.2787,Y 6.9194,Z 54,A 38.3466,B 24.7756,C -3.4526,E1 25.11,E2 -316.3107} C_DIS
LIN {X 7.2298,Y 5.9185,Z 54,A 27.7525,B 24.7795,C -3.4232,E1 25.1296,E2 -305.6943} C_DIS
LIN {X 7.9841,Y 4.8499,Z 54,A 20.4375,B 24.7816,C -3.4069,E1 25.1404,E2 -298.3775} C_DIS
LIN {X 8.7007,Y 3.4055,Z 54,A 10.8679,B 24.7848,C -3.3814,E1 25.1512,E2 -288.7996} C_DIS
LIN {X 9.1891,Y 1.6903,Z 54,A 1.1359,B 24.7881,C -3.3562,E1 25.1578,E2 -279.064} C_DIS
LIN {X 9.3145,Y 0.721,Z 54,A -5.041,B 24.7905,C -3.3368,E1 25.1596,E2 -272.8776} C_DIS
LIN {X 9.3381,Y -0.2783,Z 54,A -10.969,B 24.7928,C -3.319,E1 25.1596,E2 -266.9427} C_DIS
LIN {X 9.2407,Y -1.3751,Z 54,A -17.9721,B 24.7956,C -3.2965,E1 25.1573,E2 -259.9277} C_DIS
LIN {X 9.001,Y -2.4896,Z 54,A -24.3489,B 24.7978,C -3.2789,E1 25.1532,E2 -253.5459} C_DIS
LIN {X 8.6252,Y -3.5881,Z 54,A -30.8524,B 24.7999,C -3.2612,E1 25.147,E2 -247.037} C_DIS
LIN {X 8.2762,Y -4.3361,Z 54,A -37.3776,B 24.8028,C -3.2381,E1 25.1389,E2 -240.4918} C_DIS
LIN {X 7.5866,Y -5.4456,Z 54,A -43.2856,B 24.804,C -3.2283,E1 25.13,E2 -234.5903} C_DIS
LIN {X 7.0283,Y -6.1543,Z 54,A -50.4094,B 24.8068,C -3.2054,E1 25.1174,E2 -227.445} C_DIS
LIN {X 6.2437,Y -6.9511,Z 54,A -57.1307,B 24.8086,C -3.1902,E1 25.1039,E2 -220.7156} C_DIS
LIN {X 5.5183,Y -7.54,Z 54,A -63.0226,B 24.8101,C -3.1776,E1 25.0908,E2 -214.8152} C_DIS
LIN {X 4.3933,Y -8.2448,Z 54,A -71.3833,B 24.812,C -3.1622,E1 25.0706,E2 -206.4435} C_DIS
LIN {X 3.5756,Y -8.6306,Z 54,A -77.5957,B 24.8132,C -3.1515,E1 25.0547,E2 -200.2201} C_DIS
LIN {X 1.9152,Y -9.1433,Z 54,A -85.6261,B 24.8133,C -3.1507,E1 25.0331,E2 -192.2015} C_DIS
LIN {X 0.9999,Y -9.2883,Z 54,A -94.1849,B 24.815,C -3.1368,E1 25.0094,E2 -183.6166} C_DIS
LIN {X 0.9999,Y -9.2883,Z 54,A -94.1849,B 24.815,C -3.1368,E1 25.0094,E2 -183.6166} C_DIS
Enddeposition()
LIN {X 0.0754,Y -10.2463,Z 54,A -97.6609,B 24.8162,C -3.1265,E1 24.9996,E2 -180.1167} C_DIS
Startdeposition()
$VEL.CP = VEL_PRINT
LIN {X 0.9783,Y -10.2025,Z 54,A -90.1568,B 24.8149,C -3.1378,E1 25.0206,E2 -187.6447} C_DIS
LIN {X 1.8305,Y -10.0848,Z 54,A -85.239,B 24.8144,C -3.1419,E1 25.0341,E2 -192.567} C_DIS
LIN {X 2.792,Y -9.8618,Z 54,A -80.0566,B 24.8139,C -3.146,E1 25.0481,E2 -197.751} C_DIS
LIN {X 3.8358,Y -9.5045,Z 54,A -73.785,B 24.8129,C -3.1545,E1 25.0645,E2 -204.0296} C_DIS
LIN {X 5.1267,Y -8.8753,Z 54,A -65.9991,B 24.8115,C -3.1664,E1 25.0838,E2 -211.8219} C_DIS
LIN {X 6.0993,Y -8.2369,Z 54,A -59.2667,B 24.8098,C -3.1804,E1 25.0992,E2 -218.5645} C_DIS
LIN {X 6.9097,Y -7.5701,Z 54,A -53.4965,B 24.8083,C -3.1928,E1 25.1114,E2 -224.3414} C_DIS
LIN {X 7.6955,Y -6.7684,Z 54,A -47.3431,B 24.8065,C -3.2074,E1 25.123,E2 -230.5022} C_DIS
LIN {X 8.3419,Y -5.954,Z 54,A -41.5478,B 24.8047,C -3.2225,E1 25.1327,E2 -236.3056} C_DIS
LIN {X 8.9172,Y -5.0513,Z 54,A -35.7371,B 24.8028,C -3.238,E1 25.1411,E2 -242.1235} C_DIS
LIN {X 9.3894,Y -4.1068,Z 54,A -29.8663,B 24.8007,C -3.2549,E1 25.1481,E2 -248.0027} C_DIS
LIN {X 9.8153,Y -2.9382,Z 54,A -24.4754,B 24.7994,C -3.2659,E1 25.1531,E2 -253.3893} C_DIS
LIN {X 10.0129,Y -2.1833,Z 54,A -19.6068,B 24.7973,C -3.2824,E1 25.1564,E2 -258.269} C_DIS
LIN {X 10.1642,Y -1.3179,Z 54,A -14.2992,B 24.7951,C -3.3002,E1 25.1588,E2 -263.5875} C_DIS
LIN {X 10.2411,Y -0.4076,Z 54,A -8.4826,B 24.7925,C -3.3207,E1 25.1598,E2 -269.4182} C_DIS
LIN {X 10.2243,Y 0.6973,Z 54,A -2.6434,B 24.7904,C -3.3376,E1 25.1591,E2 -275.2628} C_DIS
LIN {X 10.1092,Y 1.6817,Z 54,A 3.1298,B 24.7881,C -3.3559,E1 25.1568,E2 -281.0455} C_DIS
LIN {X 9.7748,Y 3.0776,Z 54,A 11.3695,B 24.7849,C -3.3808,E1 25.1507,E2 -289.297} C_DIS
LIN {X 9.3883,Y 4.1095,Z 54,A 17.3099,B 24.7829,C -3.3966,E1 25.1444,E2 -295.2421} C_DIS
LIN {X 8.8404,Y 5.1868,Z 54,A 23.75,B 24.7809,C -3.4124,E1 25.1358,E2 -301.686} C_DIS
LIN {X 8.2377,Y 6.0983,Z 54,A 29.4677,B 24.7792,C -3.425,E1 25.1267,E2 -307.4055} C_DIS
LIN {X 7.6561,Y 6.814,Z 54,A 34.8079,B 24.7776,C -3.4376,E1 25.117,E2 -312.7513} C_DIS
LIN {X 6.909,Y 7.5708,Z 54,A 41.3056,B 24.7757,C -3.4524,E1 25.1039,E2 -319.2574} C_DIS
LIN {X 5.9131,Y 8.3671,Z 54,A 47.7545,B 24.7745,C -3.4613,E1 25.0896,E2 -325.7039} C_DIS
LIN {X 5.2326,Y 8.8076,Z 54,A 51.9585,B 24.7738,C -3.4663,E1 25.0796,E2 -329.9066} C_DIS
LIN {X 3.9629,Y 9.4506,Z 54,A 61.7359,B 24.7716,C -3.4835,E1 25.0549,E2 -339.6998} C_DIS
LIN {X 2.3048,Y 9.9859,Z 54,A 70.3852,B 24.7713,C -3.4853,E1 25.0317,E2 -348.3393} C_DIS
LIN {X 1.0728,Y 10.192,Z 54,A 78.233,B 24.7707,C -3.4899,E1 25.0099,E2 -356.1917} C_DIS
LIN {X -0.4556,Y 10.2396,Z 54,A 86.1276,B 24.7713,C -3.4859,E1 24.9879,E2 -364.0769} C_DIS
LIN {X -1.593,Y 10.1234,Z 54,A 91.9504,B 24.772,C -3.4806,E1 24.9718,E2 -369.8912} C_DIS
LIN {X -2.5573,Y 9.9237,Z 54,A 97.2402,B 24.7727,C -3.4753,E1 24.9574,E2 -375.1751} C_DIS
LIN {X -3.424,Y 9.6596,Z 54,A 102.838,B 24.7733,C -3.4706,E1 24.9426,E2 -380.7721} C_DIS
LIN {X -4.5096,Y 9.2009,Z 54,A 109.0801,B 24.7746,C -3.4604,E1 24.9267,E2 -387.0051} C_DIS
LIN {X -5.5663,Y 8.6058,Z 54,A 116.1497,B 24.7761,C -3.449,E1 24.9098,E2 -394.0687} C_DIS
LIN {X -6.4375,Y 7.9754,Z 54,A 122.9159,B 24.7776,C -3.4377,E1 24.8949,E2 -400.8326} C_DIS
LIN {X -7.7058,Y 6.7564,Z 54,A 133.0111,B 24.7806,C -3.4147,E1 24.8754,E2 -410.9162} C_DIS
LIN {X -8.6109,Y 5.5592,Z 54,A 140.22,B 24.7835,C -3.3916,E1 24.8638,E2 -418.1052} C_DIS
LIN {X -9.1505,Y 4.6159,Z 54,A 146.8795,B 24.7857,C -3.3748,E1 24.855,E2 -424.7596} C_DIS
LIN {X -9.586,Y 3.624,Z 54,A 152.8171,B 24.788,C -3.357,E1 24.8487,E2 -430.6875} C_DIS
LIN {X -9.9039,Y 2.6331,Z 54,A 158.4641,B 24.7902,C -3.3393,E1 24.8443,E2 -436.3247} C_DIS
LIN {X -10.1126,Y 1.6602,Z 54,A 164.7612,B 24.7923,C -3.3224,E1 24.8411,E2 -442.6185} C_DIS
LIN {X -10.2417,Y 0.4001,Z 54,A 171.1905,B 24.7951,C -3.3002,E1 24.8398,E2 -449.0333} C_DIS
LIN {X -10.2344,Y -0.5474,Z 54,A 176.5133,B 24.7971,C -3.2839,E1 24.8402,E2 -454.3489} C_DIS
LIN {X -10.0175,Y -2.1617,Z 54,A -172.3692,B 24.8004,C -3.2572,E1 24.8455,E2 -465.4685} C_DIS
LIN {X -9.4967,Y -3.8544,Z 54,A -163.5846,B 24.804,C -3.2284,E1 24.8538,E2 -474.2336} C_DIS
LIN {X -9.0012,Y -4.8983,Z 54,A -157.666,B 24.8061,C -3.2108,E1 24.8613,E2 -480.1419} C_DIS
LIN {X -8.467,Y -5.773,Z 54,A -152.2177,B 24.8079,C -3.1963,E1 24.8695,E2 -485.5829} C_DIS
LIN {X -7.7957,Y -6.6513,Z 54,A -146.098,B 24.8096,C -3.1821,E1 24.8801,E2 -491.6973} C_DIS
LIN {X -7.1163,Y -7.3717,Z 54,A -140.2886,B 24.8109,C -3.171,E1 24.8914,E2 -497.5051} C_DIS
LIN {X -6.373,Y -8.0263,Z 54,A -134.1371,B 24.812,C -3.1619,E1 24.9046,E2 -503.6584} C_DIS
LIN {X -5.2797,Y -8.7838,Z 54,A -128.2538,B 24.8137,C -3.1477,E1 24.9183,E2 -509.527} C_DIS
LIN {X -4.6452,Y -9.1361,Z 54,A -122.4323,B 24.8139,C -3.1463,E1 24.9327,E2 -515.3615} C_DIS
LIN {X -3.6637,Y -9.5714,Z 54,A -116.84,B 24.8147,C -3.1396,E1 24.9471,E2 -520.9501} C_DIS
LIN {X -2.4625,Y -9.9454,Z 54,A -111.3788,B 24.8157,C -3.1306,E1 24.9617,E2 -526.3992} C_DIS
LIN {X -1.6775,Y -10.1099,Z 54,A -106.074,B 24.8157,C -3.1313,E1 24.9762,E2 -531.7116} C_DIS
LIN {X -0.7931,Y -10.2179,Z 54,A -100.3431,B 24.8154,C -3.1334,E1 24.9922,E2 -537.4505} C_DIS
LIN {X 0.0754,Y -10.2463,Z 54,A -97.6609,B 24.8162,C -3.1265,E1 24.9996,E2 -540.1167} C_DIS
Enddeposition()
LIN {X 0.0754,Y -10.2463,Z 54,A -97.6609,B 24.8162,C -3.1265,E1 24.9996,E2 -540.1167} C_DIS
Startdeposition()
$VEL.CP = VEL_PRINT
LIN {X -0.4528,Y -11.1436,Z 54,A -100.4591,B 24.8181,C -3.11,E1 24.9917,E2 -537.2789} C_DIS
LIN {X -1.3376,Y -11.074,Z 54,A -105.6717,B 24.8184,C -3.1081,E1 24.9772,E2 -532.0588} C_DIS
LIN {X -2.5369,Y -10.8637,Z 54,A -111.7724,B 24.818,C -3.111,E1 24.9605,E2 -525.9581} C_DIS
LIN {X -3.6641,Y -10.5367,Z 54,A -117.6189,B 24.8175,C -3.1158,E1 24.9449,E2 -520.1128} C_DIS
LIN {X -4.5295,Y -10.1944,Z 54,A -123.1622,B 24.8171,C -3.1186,E1 24.9307,E2 -514.5635} C_DIS
LIN {X -5.7446,Y -9.5617,Z 54,A -129.4725,B 24.8159,C -3.1294,E1 24.9153,E2 -508.2608} C_DIS
LIN {X -6.4395,Y -9.1079,Z 54,A -134.0593,B 24.8151,C -3.1355,E1 24.9047,E2 -503.6731} C_DIS
LIN {X -7.241,Y -8.4838,Z 54,A -139.1768,B 24.814,C -3.145,E1 24.8936,E2 -498.559} C_DIS
LIN {X -8.2192,Y -7.5422,Z 54,A -146.7649,B 24.8124,C -3.1584,E1 24.8788,E2 -490.9707} C_DIS
LIN {X -8.9637,Y -6.6407,Z 54,A -152.8218,B 24.8108,C -3.1722,E1 24.8684,E2 -484.9182} C_DIS
LIN {X -9.7058,Y -5.4938,Z 54,A -158.2546,B 24.8084,C -3.1915,E1 24.8604,E2 -479.5039} C_DIS
LIN {X -10.0624,Y -4.8127,Z 54,A -163.2942,B 24.8073,C -3.2011,E1 24.8541,E2 -474.4602} C_DIS
LIN {X -10.4903,Y -3.7904,Z 54,A -169.4582,B 24.8054,C -3.2168,E1 24.8478,E2 -468.2992} C_DIS
LIN {X -10.8924,Y -2.4047,Z 54,A -177.125,B 24.8027,C -3.2385,E1 24.8425,E2 -460.6398} C_DIS
LIN {X -11.0894,Y -1.2023,Z 54,A 177.1012,B 24.8004,C -3.2577,E1 24.8404,E2 -454.8777} C_DIS
LIN {X -11.1527,Y -0.1154,Z 54,A 171.7393,B 24.7982,C -3.2751,E1 24.8398,E2 -449.5252} C_DIS
LIN {X -11.1256,Y 0.8011,Z 54,A 166.6684,B 24.7964,C -3.2896,E1 24.8405,E2 -444.4584} C_DIS
LIN {X -10.9861,Y 1.936,Z 54,A 160.8051,B 24.7942,C -3.3077,E1 24.8429,E2 -438.6037} C_DIS
LIN {X -10.7397,Y 3.0182,Z 54,A 154.8172,B 24.792,C -3.325,E1 24.847,E2 -432.6223} C_DIS
LIN {X -10.3758,Y 4.0985,Z 54,A 149.2441,B 24.7898,C -3.3425,E1 24.8524,E2 -427.0598} C_DIS
LIN {X -9.9252,Y 5.0935,Z 54,A 143.5224,B 24.7877,C -3.3586,E1 24.8593,E2 -421.3457} C_DIS
LIN {X -9.3399,Y 6.1009,Z 54,A 137.0748,B 24.7857,C -3.3747,E1 24.8687,E2 -414.9035} C_DIS
LIN {X -8.5474,Y 7.1638,Z 54,A 130.7667,B 24.7834,C -3.3926,E1 24.8795,E2 -408.6086} C_DIS
LIN {X -7.5926,Y 8.1713,Z 54,A 123.4808,B 24.7813,C -3.4091,E1 24.8938,E2 -401.3312} C_DIS
LIN {X -6.7691,Y 8.865,Z 54,A 117.5269,B 24.7799,C -3.42,E1 24.9068,E2 -395.3813} C_DIS
LIN {X -5.6962,Y 9.5915,Z 54,A 111.1678,B 24.7782,C -3.4326,E1 24.9218,E2 -389.0321} C_DIS
LIN {X -4.6575,Y 10.1371,Z 54,A 105.2275,B 24.777,C -3.4421,E1 24.9366,E2 -383.0988} C_DIS
LIN {X -3.6827,Y 10.5299,Z 54,A 99.5584,B 24.7762,C -3.4484,E1 24.9514,E2 -377.4329} C_DIS
LIN {X -2.6921,Y 10.825,Z 54,A 94.2291,B 24.7755,C -3.4536,E1 24.9658,E2 -372.108} C_DIS
LIN {X -1.7119,Y 11.0222,Z 54,A 89.3318,B 24.7749,C -3.458,E1 24.9792,E2 -367.2163} C_DIS
LIN {X -0.6549,Y 11.1354,Z 54,A 83.9297,B 24.7746,C -3.4606,E1 24.9942,E2 -361.818} C_DIS
LIN {X 0.4918,Y 11.1451,Z 54,A 78.0116,B 24.7745,C -3.4614,E1 25.0107,E2 -355.9024} C_DIS
LIN {X 1.812,Y 11.0061,Z 54,A 70.7706,B 24.7749,C -3.4584,E1 25.0308,E2 -348.6603} C_DIS
LIN {X 3.1344,Y 10.7063,Z 54,A 64.4114,B 24.7751,C -3.4569,E1 25.048,E2 -342.3069} C_DIS
LIN {X 4.03,Y 10.4022,Z 54,A 59.176,B 24.7758,C -3.451,E1 25.0617,E2 -337.0683} C_DIS
LIN {X 5.0283,Y 9.9576,Z 54,A 53.3512,B 24.7768,C -3.4435,E1 25.0764,E2 -331.2409} C_DIS
LIN {X 6.2715,Y 9.224,Z 54,A 45.8995,B 24.7783,C -3.4323,E1 25.094,E2 -323.7865} C_DIS
LIN {X 6.9863,Y 8.6972,Z 54,A 41.1881,B 24.7794,C -3.4235,E1 25.1043,E2 -319.0715} C_DIS
LIN {X 8.2239,Y 7.5373,Z 54,A 32.9664,B 24.7814,C -3.4084,E1 25.1206,E2 -310.8487} C_DIS
LIN {X 9.0227,Y 6.5609,Z 54,A 26.3136,B 24.7834,C -3.3923,E1 25.132,E2 -304.1891} C_DIS
LIN {X 9.562,Y 5.7442,Z 54,A 21.2905,B 24.7851,C -3.3796,E1 25.1394,E2 -299.1614} C_DIS
LIN {X 10.1851,Y 4.5511,Z 54,A 15.0713,B 24.7869,C -3.3653,E1 25.147,E2 -292.9415} C_DIS
LIN {X 10.5487,Y 3.6301,Z 54,A 9.5934,B 24.789,C -3.3484,E1 25.1524,E2 -287.454} C_DIS
LIN {X 10.8322,Y 2.6642,Z 54,A 4.104,B 24.7912,C -3.3311,E1 25.1563,E2 -281.9552} C_DIS
LIN {X 11.07,Y 1.3518,Z 54,A -1.976,B 24.7932,C -3.3155,E1 25.1589,E2 -275.8738} C_DIS
LIN {X 11.1496,Y 0.3345,Z 54,A -7.6383,B 24.7956,C -3.2965,E1 25.1598,E2 -270.2001} C_DIS
LIN {X 11.1207,Y -0.8484,Z 54,A -13.1462,B 24.7974,C -3.2814,E1 25.1591,E2 -264.6893} C_DIS
LIN {X 11.0019,Y -1.8377,Z 54,A -18.8717,B 24.7999,C -3.2615,E1 25.1568,E2 -258.9502} C_DIS
LIN {X 10.7641,Y -2.9258,Z 54,A -24.3415,B 24.8019,C -3.2456,E1 25.1531,E2 -253.4744} C_DIS
LIN {X 10.3607,Y -4.1365,Z 54,A -30.7011,B 24.8041,C -3.2272,E1 25.1471,E2 -247.1069} C_DIS
LIN {X 9.8469,Y -5.2411,Z 54,A -36.6191,B 24.806,C -3.2114,E1 25.1398,E2 -241.183} C_DIS
LIN {X 9.3691,Y -6.0556,Z 54,A -42.4001,B 24.8084,C -3.1921,E1 25.1313,E2 -235.3857} C_DIS
LIN {X 8.5241,Y -7.1924,Z 54,A -47.863,B 24.8093,C -3.1845,E1 25.122,E2 -229.9305} C_DIS
LIN {X 7.9918,Y -7.7818,Z 54,A -53.2201,B 24.8114,C -3.1669,E1 25.1118,E2 -224.5551} C_DIS
LIN {X 7.1069,Y -8.5984,Z 54,A -59.5607,B 24.8131,C -3.1523,E1 25.0984,E2 -218.2048} C_DIS
LIN {X 5.9619,Y -9.4275,Z 54,A -65.7629,B 24.8141,C -3.144,E1 25.0842,E2 -212.0041} C_DIS
LIN {X 5.1784,Y -9.881,Z 54,A -71.4182,B 24.8157,C -3.1308,E1 25.0704,E2 -206.3339} C_DIS
LIN {X 4.0345,Y -10.4005,Z 54,A -77.1985,B 24.8164,C -3.1249,E1 25.0555,E2 -200.5535} C_DIS
LIN {X 2.9789,Y -10.7499,Z 54,A -83.7491,B 24.8176,C -3.1146,E1 25.038,E2 -193.99} C_DIS
LIN {X 1.7601,Y -11.0144,Z 54,A -89.8406,B 24.818,C -3.1109,E1 25.0213,E2 -187.8966} C_DIS
LIN {X 0.8496,Y -11.1223,Z 54,A -94.3648,B 24.8182,C -3.1092,E1 25.0087,E2 -183.3711} C_DIS
LIN {X 0.0798,Y -11.151,Z 54,A -97.1076,B 24.8178,C -3.1128,E1 25.0011,E2 -180.6373} C_DIS
Enddeposition()
LIN {X 0.0798,Y -11.151,Z 54,A -97.1076,B 24.8178,C -3.1128,E1 25.0011,E2 -180.6373} C_DIS
Startdeposition()
$VEL.CP = VEL_PRINT
LIN {X 0.6754,Y -12.0404,Z 54,A -93.1432,B 24.819,C -3.103,E1 25.0121,E2 -184.5774} C_DIS
LIN {X 1.7686,Y -11.9309,Z 54,A -87.7892,B 24.8185,C -3.1067,E1 25.0269,E2 -189.9361} C_DIS
LIN {X 2.7719,Y -11.7393,Z 54,A -82.8658,B 24.818,C -3.1113,E1 25.0404,E2 -194.8641} C_DIS
LIN {X 3.6932,Y -11.4812,Z 54,A -78.2607,B 24.8174,C -3.1167,E1 25.0527,E2 -199.4739} C_DIS
LIN {X 4.6783,Y -11.1158,Z 54,A -73.3568,B 24.8166,C -3.123,E1 25.0654,E2 -204.3819} C_DIS
LIN {X 5.6229,Y -10.6709,Z 54,A -68.1962,B 24.8156,C -3.132,E1 25.0783,E2 -209.5498} C_DIS
LIN {X 6.6865,Y -10.0386,Z 54,A -62.2284,B 24.8142,C -3.1434,E1 25.0924,E2 -215.5255} C_DIS
LIN {X 7.5676,Y -9.3928,Z 54,A -57.1518,B 24.813,C -3.1535,E1 25.1036,E2 -220.6074} C_DIS
LIN {X 8.5739,Y -8.4841,Z 54,A -50.7944,B 24.8113,C -3.1678,E1 25.1165,E2 -226.9725} C_DIS
LIN {X 9.3176,Y -7.6597,Z 54,A -45.6112,B 24.8098,C -3.1804,E1 25.126,E2 -232.1621} C_DIS
LIN {X 9.8783,Y -6.9186,Z 54,A -41.4969,B 24.8086,C -3.1901,E1 25.1327,E2 -236.2796} C_DIS
LIN {X 10.4281,Y -6.0622,Z 54,A -36.5207,B 24.8069,C -3.2044,E1 25.14,E2 -241.2642} C_DIS
LIN {X 10.9012,Y -5.1597,Z 54,A -31.9112,B 24.8054,C -3.2167,E1 25.1457,E2 -245.8785} C_DIS
LIN {X 11.2661,Y -4.3066,Z 54,A -27.4694,B 24.8038,C -3.23,E1 25.1504,E2 -250.3272} C_DIS
LIN {X 11.5901,Y -3.3413,Z 54,A -22.5209,B 24.8019,C -3.2454,E1 25.1545,E2 -255.2842} C_DIS
LIN {X 11.8109,Y -2.4401,Z 54,A -18.0249,B 24.8001,C -3.2597,E1 25.1572,E2 -259.7878} C_DIS
LIN {X 11.9893,Y -1.309,Z 54,A -12.6805,B 24.7981,C -3.2759,E1 25.1592,E2 -265.1391} C_DIS
LIN {X 12.0615,Y -0.0862,Z 54,A -6.8429,B 24.7959,C -3.2941,E1 25.1597,E2 -270.9851} C_DIS
LIN {X 12.019,Y 1.017,Z 54,A -1.7551,B 24.794,C -3.3091,E1 25.1589,E2 -276.0784} C_DIS
LIN {X 11.8893,Y 2.0273,Z 54,A 2.8588,B 24.7923,C -3.3223,E1 25.157,E2 -280.6963} C_DIS
LIN {X 11.6982,Y 2.9346,Z 54,A 7.2883,B 24.7907,C -3.3355,E1 25.1542,E2 -285.1316} C_DIS
LIN {X 11.4072,Y 3.9204,Z 54,A 12.2292,B 24.7888,C -3.35,E1 25.15,E2 -290.0788} C_DIS
LIN {X 11.0704,Y 4.7851,Z 54,A 16.9951,B 24.787,C -3.3648,E1 25.1449,E2 -294.8535} C_DIS
LIN {X 10.426,Y 6.0658,Z 54,A 23.5964,B 24.7849,C -3.3813,E1 25.1361,E2 -301.4593} C_DIS
LIN {X 9.8764,Y 6.9215,Z 54,A 28.2099,B 24.7835,C -3.3918,E1 25.1289,E2 -306.0749} C_DIS
LIN {X 9.2585,Y 7.7294,Z 54,A 32.8623,B 24.7822,C -3.4018,E1 25.1208,E2 -310.7293} C_DIS
LIN {X 8.4801,Y 8.5777,Z 54,A 38.3939,B 24.7807,C -3.4136,E1 25.1101,E2 -316.2652} C_DIS
LIN {X 7.4895,Y 9.454,Z 54,A 44.5759,B 24.7793,C -3.4247,E1 25.097,E2 -322.4495} C_DIS
LIN {X 6.6677,Y 10.0513,Z 54,A 49.6416,B 24.7781,C -3.4338,E1 25.0854,E2 -327.5194} C_DIS
LIN {X 5.8736,Y 10.5333,Z 54,A 53.7783,B 24.7775,C -3.4385,E1 25.0754,E2 -331.6548} C_DIS
LIN {X 4.9685,Y 10.9913,Z 54,A 58.7286,B 24.7767,C -3.4447,E1 25.0629,E2 -336.607} C_DIS
LIN {X 4.0254,Y 11.3694,Z 54,A 63.8185,B 24.7759,C -3.4504,E1 25.0496,E2 -341.6995} C_DIS
LIN {X 2.6366,Y 11.7697,Z 54,A 70.3214,B 24.7756,C -3.4528,E1 25.032,E2 -348.1982} C_DIS
LIN {X 1.6358,Y 11.9507,Z 54,A 75.1328,B 24.7754,C -3.4542,E1 25.0188,E2 -353.008} C_DIS
LIN {X 0.4774,Y 12.0525,Z 54,A 81.29,B 24.7751,C -3.4567,E1 25.0016,E2 -359.1687} C_DIS
LIN {X -0.8156,Y 12.0329,Z 54,A 86.5948,B 24.7757,C -3.4518,E1 24.9868,E2 -364.4627} C_DIS
LIN {X -1.7371,Y 11.9359,Z 54,A 91.255,B 24.776,C -3.4501,E1 24.9739,E2 -369.1222} C_DIS
LIN {X -2.7366,Y 11.7476,Z 54,A 96.204,B 24.7764,C -3.4464,E1 24.9604,E2 -374.0684} C_DIS
LIN {X -3.6297,Y 11.5011,Z 54,A 100.5534,B 24.7771,C -3.4416,E1 24.9488,E2 -378.4136} C_DIS
LIN {X -4.586,Y 11.1551,Z 54,A 105.2946,B 24.7779,C -3.4351,E1 24.9365,E2 -383.1493} C_DIS
LIN {X -5.511,Y 10.7296,Z 54,A 110.294,B 24.7788,C -3.4281,E1 24.9239,E2 -388.1449} C_DIS
LIN {X -6.3169,Y 10.2733,Z 54,A 114.6025,B 24.7798,C -3.4203,E1 24.9136,E2 -392.4477} C_DIS
LIN {X -7.1625,Y 9.7051,Z 54,A 119.5664,B 24.781,C -3.4111,E1 24.9023,E2 -397.4067} C_DIS
LIN {X -7.9023,Y 9.1106,Z 54,A 124.1054,B 24.7823,C -3.4015,E1 24.8926,E2 -401.9402} C_DIS
LIN {X -8.6431,Y 8.4119,Z 54,A 128.8043,B 24.7837,C -3.3901,E1 24.8832,E2 -406.6315} C_DIS
LIN {X -9.3216,Y 7.6549,Z 54,A 133.9437,B 24.7852,C -3.3786,E1 24.8739,E2 -411.7667} C_DIS
LIN {X -9.8831,Y 6.9117,Z 54,A 138.1232,B 24.7867,C -3.3667,E1 24.8671,E2 -415.938} C_DIS
LIN {X -10.4316,Y 6.0562,Z 54,A 143.1462,B 24.7884,C -3.3536,E1 24.8598,E2 -420.9554} C_DIS
LIN {X -10.9035,Y 5.1552,Z 54,A 147.8319,B 24.7902,C -3.3397,E1 24.8539,E2 -425.6329} C_DIS
LIN {X -11.2675,Y 4.3027,Z 54,A 152.3117,B 24.7918,C -3.3268,E1 24.8493,E2 -430.1068} C_DIS
LIN {X -11.5906,Y 3.3398,Z 54,A 157.3237,B 24.7936,C -3.3124,E1 24.8451,E2 -435.113} C_DIS
LIN {X -11.8399,Y 2.302,Z 54,A 162.2331,B 24.7955,C -3.2967,E1 24.8422,E2 -440.0137} C_DIS
LIN {X -11.9746,Y 1.4381,Z 54,A 166.5227,B 24.7971,C -3.2839,E1 24.8406,E2 -444.2984} C_DIS
LIN {X -12.0566,Y 0.3114,Z 54,A 171.2002,B 24.7993,C -3.2667,E1 24.8398,E2 -448.9627} C_DIS
LIN {X -12.0503,Y -0.5344,Z 54,A 176.0372,B 24.8007,C -3.255,E1 24.8401,E2 -453.8006} C_DIS
LIN {X -11.962,Y -1.5481,Z 54,A -179.032,B 24.8025,C -3.2403,E1 24.8416,E2 -458.7257} C_DIS
LIN {X -11.806,Y -2.4638,Z 54,A -174.6978,B 24.8041,C -3.227,E1 24.8439,E2 -463.0537} C_DIS
LIN {X -11.5607,Y -3.439,Z 54,A -169.6689,B 24.8058,C -3.2132,E1 24.8476,E2 -468.0788} C_DIS
LIN {X -11.2345,Y -4.3907,Z 54,A -164.8516,B 24.8075,C -3.1997,E1 24.8523,E2 -472.891} C_DIS
LIN {X -10.8998,Y -5.1627,Z 54,A -160.7963,B 24.8088,C -3.1889,E1 24.857,E2 -476.9425} C_DIS
LIN {X -10.38,Y -6.1436,Z 54,A -155.7299,B 24.8104,C -3.1749,E1 24.864,E2 -482.0019} C_DIS
LIN {X -9.8758,Y -6.9223,Z 54,A -151.031,B 24.8117,C -3.1646,E1 24.8713,E2 -486.6996} C_DIS
LIN {X -9.2465,Y -7.7435,Z 54,A -146.4792,B 24.8131,C -3.1528,E1 24.8793,E2 -491.2443} C_DIS
LIN {X -8.5647,Y -8.4935,Z 54,A -141.3501,B 24.8142,C -3.1433,E1 24.8891,E2 -496.3729} C_DIS
LIN {X -7.8854,Y -9.125,Z 54,A -137.1921,B 24.8153,C -3.1344,E1 24.8978,E2 -500.5263} C_DIS
LIN {X -7.0931,Y -9.7562,Z 54,A -132.1839,B 24.8162,C -3.1266,E1 24.9089,E2 -505.534} C_DIS
LIN {X -6.2394,Y -10.3212,Z 54,A -127.5128,B 24.8171,C -3.119,E1 24.9199,E2 -510.2018} C_DIS
LIN {X -5.4276,Y -10.7712,Z 54,A -123.0053,B 24.8177,C -3.1138,E1 24.931,E2 -514.7092} C_DIS
LIN {X -4.5003,Y -11.191,Z 54,A -117.674,B 24.8181,C -3.1104,E1 24.9447,E2 -520.0447} C_DIS
LIN {X -3.1369,Y -11.6456,Z 54,A -111.3198,B 24.8188,C -3.1041,E1 24.9617,E2 -526.3948} C_DIS
LIN {X -2.1443,Y -11.8699,Z 54,A -106.4032,B 24.819,C -3.1024,E1 24.9751,E2 -531.3132} C_DIS
LIN {X -1.2257,Y -11.9987,Z 54,A -101.9409,B 24.819,C -3.102,E1 24.9875,E2 -535.7775} C_DIS
LIN {X -0.2095,Y -12.0588,Z 54,A -96.8419,B 24.8189,C -3.1037,E1 25.0018,E2 -540.8813} C_DIS
LIN {X -0.2095,Y -12.0588,Z 54,A -96.8419,B 24.8189,C -3.1037,E1 25.0018,E2 -540.8813} C_DIS
Enddeposition()
LIN {X 0.0449,Y -12.4206,Z 55,A -97.0281,B 24.8195,C -3.0985,E1 25.0012,E2 -540.6828} C_DIS
Startdeposition()
$VEL.CP = VEL_PRINT
LIN {X -0.9751,Y -12.3871,Z 55,A -103.4379,B 24.8204,C -3.0911,E1 24.9833,E2 -534.2538} C_DIS
LIN {X -2.261,Y -12.218,Z 55,A -109.2471,B 24.8201,C -3.0933,E1 24.9673,E2 -528.4446} C_DIS
LIN {X -3.532,Y -11.9127,Z 55,A -115.2801,B 24.8197,C -3.0968,E1 24.951,E2 -522.4108} C_DIS
LIN {X -4.717,Y -11.4953,Z 55,A -121.0559,B 24.8191,C -3.102,E1 24.9359,E2 -516.6354} C_DIS
LIN {X -5.8244,Y -10.9757,Z 55,A -126.8657,B 24.8184,C -3.1083,E1 24.9214,E2 -510.825} C_DIS
LIN {X -6.998,Y -10.2674,Z 55,A -133.3029,B 24.8173,C -3.1174,E1 24.9063,E2 -504.389} C_DIS
LIN {X -8.0688,Y -9.4491,Z 55,A -139.397,B 24.8159,C -3.1287,E1 24.8931,E2 -498.299} C_DIS
LIN {X -9.0019,Y -8.5648,Z 55,A -145.3563,B 24.8145,C -3.1407,E1 24.8813,E2 -492.3432} C_DIS
LIN {X -9.8377,Y -7.5902,Z 55,A -151.3292,B 24.8129,C -3.1541,E1 24.8708,E2 -486.3746} C_DIS
LIN {X -10.6055,Y -6.4741,Z 55,A -157.5989,B 24.8111,C -3.1695,E1 24.8612,E2 -480.1103} C_DIS
LIN {X -11.2306,Y -5.3162,Z 55,A -163.7206,B 24.8092,C -3.1856,E1 24.8535,E2 -473.9944} C_DIS
LIN {X -11.7421,Y -4.0633,Z 55,A -170.0433,B 24.807,C -3.2032,E1 24.8473,E2 -467.6782} C_DIS
LIN {X -12.1019,Y -2.8167,Z 55,A -176.1309,B 24.8049,C -3.2207,E1 24.843,E2 -461.5971} C_DIS
LIN {X -12.3399,Y -1.443,Z 55,A 178.392,B 24.8024,C -3.2411,E1 24.8407,E2 -456.1363} C_DIS
LIN {X -12.4335,Y -0.0382,Z 55,A 172.8002,B 24.7999,C -3.2617,E1 24.8398,E2 -450.5604} C_DIS
LIN {X -12.3926,Y 0.8995,Z 55,A 167.9357,B 24.7983,C -3.2748,E1 24.8402,E2 -445.6979} C_DIS
LIN {X -12.2508,Y 2.0749,Z 55,A 161.1414,B 24.7963,C -3.2906,E1 24.8427,E2 -438.901} C_DIS
LIN {X -11.9683,Y 3.3384,Z 55,A 154.9923,B 24.794,C -3.3087,E1 24.8469,E2 -432.7593} C_DIS
LIN {X -11.553,Y 4.5737,Z 55,A 149.1239,B 24.7918,C -3.3267,E1 24.8525,E2 -426.901} C_DIS
LIN {X -11.0373,Y 5.7069,Z 55,A 143.2733,B 24.7897,C -3.3431,E1 24.8596,E2 -421.0581} C_DIS
LIN {X -10.3631,Y 6.8554,Z 55,A 137.0457,B 24.7876,C -3.3598,E1 24.8688,E2 -414.8387} C_DIS
LIN {X -9.5958,Y 7.8938,Z 55,A 131.0373,B 24.7857,C -3.375,E1 24.8791,E2 -408.8383} C_DIS
LIN {X -8.6806,Y 8.8903,Z 55,A 124.791,B 24.7838,C -3.3897,E1 24.8912,E2 -402.6004} C_DIS
LIN {X -7.7066,Y 9.7468,Z 55,A 118.7841,B 24.7821,C -3.4025,E1 24.9041,E2 -396.601} C_DIS
LIN {X -6.6306,Y 10.5083,Z 55,A 112.6095,B 24.7807,C -3.4137,E1 24.9184,E2 -390.4328} C_DIS
LIN {X -5.4267,Y 11.1778,Z 55,A 106.379,B 24.7793,C -3.4242,E1 24.9338,E2 -384.2103} C_DIS
LIN {X -4.2863,Y 11.6627,Z 55,A 100.6301,B 24.7784,C -3.4317,E1 24.9487,E2 -378.4667} C_DIS
LIN {X -3.1291,Y 12.025,Z 55,A 95.0571,B 24.7776,C -3.4375,E1 24.9636,E2 -372.8988} C_DIS
LIN {X -1.8518,Y 12.2866,Z 55,A 89.0351,B 24.777,C -3.442,E1 24.9801,E2 -366.8811} C_DIS
LIN {X -0.5539,Y 12.4131,Z 55,A 82.7892,B 24.7768,C -3.4436,E1 24.9975,E2 -360.6368} C_DIS
LIN {X 0.8278,Y 12.3978,Z 55,A 76.3966,B 24.7768,C -3.444,E1 25.0153,E2 -354.2468} C_DIS
LIN {X 2.1393,Y 12.2398,Z 55,A 70.3231,B 24.777,C -3.4425,E1 25.0321,E2 -348.1752} C_DIS
LIN {X 3.4661,Y 11.932,Z 55,A 64.0662,B 24.7774,C -3.4388,E1 25.049,E2 -341.9194} C_DIS
LIN {X 4.717,Y 11.4953,Z 55,A 58.1522,B 24.778,C -3.4342,E1 25.0644,E2 -336.0069} C_DIS
LIN {X 5.8461,Y 10.9642,Z 55,A 52.1909,B 24.7791,C -3.4261,E1 25.0793,E2 -330.0426} C_DIS
LIN {X 6.998,Y 10.2674,Z 55,A 45.9834,B 24.7803,C -3.4167,E1 25.0939,E2 -323.833} C_DIS
LIN {X 8.0956,Y 9.4261,Z 55,A 39.6516,B 24.7817,C -3.4055,E1 25.1076,E2 -317.4984} C_DIS
LIN {X 9.069,Y 8.4937,Z 55,A 33.4455,B 24.7834,C -3.3927,E1 25.1198,E2 -311.2885} C_DIS
LIN {X 9.9422,Y 7.4528,Z 55,A 27.2095,B 24.7852,C -3.3785,E1 25.1306,E2 -305.0478} C_DIS
LIN {X 10.6998,Y 6.317,Z 55,A 20.9734,B 24.7872,C -3.363,E1 25.1399,E2 -298.8064} C_DIS
LIN {X 11.3106,Y 5.1442,Z 55,A 15.1275,B 24.7891,C -3.3482,E1 25.147,E2 -292.9568} C_DIS
LIN {X 11.7647,Y 3.9979,Z 55,A 9.4648,B 24.7911,C -3.3322,E1 25.1525,E2 -287.2877} C_DIS
LIN {X 12.1019,Y 2.8167,Z 55,A 3.6456,B 24.7933,C -3.3144,E1 25.1566,E2 -281.46} C_DIS
LIN {X 12.3422,Y 1.4225,Z 55,A -1.691,B 24.7948,C -3.303,E1 25.1589,E2 -276.1276} C_DIS
LIN {X 12.4323,Y 0.0515,Z 55,A -6.7452,B 24.7961,C -3.2924,E1 25.1597,E2 -271.0784} C_DIS
LIN {X 12.4131,Y -0.5539,Z 55,A -11.8914,B 24.7992,C -3.2671,E1 25.1594,E2 -265.9027} C_DIS
LIN {X 12.2747,Y -1.9283,Z 55,A -18.1372,B 24.8015,C -3.2482,E1 25.1572,E2 -259.6489} C_DIS
LIN {X 11.9924,Y -3.2514,Z 55,A -24.2253,B 24.8038,C -3.2301,E1 25.1532,E2 -253.5531} C_DIS
LIN {X 11.6173,Y -4.4077,Z 55,A -29.8684,B 24.8058,C -3.213,E1 25.148,E2 -247.9012} C_DIS
LIN {X 11.1085,Y -5.5671,Z 55,A -35.8047,B 24.808,C -3.1954,E1 25.1409,E2 -241.9552} C_DIS
LIN {X 10.4366,Y -6.743,Z 55,A -42.0277,B 24.81,C -3.1783,E1 25.1318,E2 -235.7233} C_DIS
LIN {X 9.6386,Y -7.8414,Z 55,A -48.2387,B 24.812,C -3.1623,E1 25.1212,E2 -229.5039} C_DIS
LIN {X 8.738,Y -8.834,Z 55,A -54.3408,B 24.8137,C -3.148,E1 25.1094,E2 -223.3942} C_DIS
LIN {X 7.7066,Y -9.7468,Z 55,A -60.5781,B 24.8152,C -3.1349,E1 25.0961,E2 -217.1499} C_DIS
LIN {X 6.609,Y -10.522,Z 55,A -66.7592,B 24.8166,C -3.1232,E1 25.0817,E2 -210.9615} C_DIS
LIN {X 5.4267,Y -11.1778,Z 55,A -72.8805,B 24.8177,C -3.1136,E1 25.0666,E2 -204.8346} C_DIS
LIN {X 4.2863,Y -11.6627,Z 55,A -78.5931,B 24.8186,C -3.1059,E1 25.0517,E2 -199.1164} C_DIS
LIN {X 3.1291,Y -12.025,Z 55,A -84.2013,B 24.8194,C -3.0998,E1 25.0367,E2 -193.5031} C_DIS
LIN {X 1.8294,Y -12.29,Z 55,A -90.527,B 24.82,C -3.0941,E1 25.0193,E2 -187.1708} C_DIS
LIN {X 0.4146,Y -12.4185,Z 55,A -97.0118,B 24.8203,C -3.0917,E1 25.0012,E2 -180.6828} C_DIS
LIN {X 0.4146,Y -12.4185,Z 55,A -97.0118,B 24.8203,C -3.0917,E1 25.0012,E2 -180.6828} C_DIS
Enddeposition()
LIN {X 0.064,Y -11.4666,Z 55,A -95.9933,B 24.8171,C -3.1187,E1 25.0042,E2 -181.7656} C_DIS
Startdeposition()
$VEL.CP = VEL_PRINT
LIN {X 1.0672,Y -11.4143,Z 55,A -90.9988,B 24.8169,C -3.1209,E1 25.0181,E2 -186.7631} C_DIS
LIN {X 1.8642,Y -11.3113,Z 55,A -87.1725,B 24.8167,C -3.1227,E1 25.0287,E2 -190.5903} C_DIS
LIN {X 3.1844,Y -11.0156,Z 55,A -79.2838,B 24.8152,C -3.1348,E1 25.0501,E2 -198.4957} C_DIS
LIN {X 4.5377,Y -10.5306,Z 55,A -73.6704,B 24.8151,C -3.1362,E1 25.0647,E2 -204.1003} C_DIS
LIN {X 5.4823,Y -10.0713,Z 55,A -66.9632,B 24.8131,C -3.1526,E1 25.0814,E2 -210.8281} C_DIS
LIN {X 6.579,Y -9.3919,Z 55,A -61.1579,B 24.8121,C -3.1612,E1 25.0949,E2 -216.6344} C_DIS
LIN {X 7.4549,Y -8.7128,Z 55,A -55.3766,B 24.8105,C -3.1745,E1 25.1075,E2 -222.4253} C_DIS
LIN {X 8.4158,Y -7.7848,Z 55,A -50.3537,B 24.8098,C -3.18,E1 25.1174,E2 -227.4402} C_DIS
LIN {X 8.9398,Y -7.1812,Z 55,A -45.373,B 24.8079,C -3.1962,E1 25.1264,E2 -232.4366} C_DIS
LIN {X 9.4836,Y -6.4459,Z 55,A -40.1758,B 24.8059,C -3.2124,E1 25.1348,E2 -237.647} C_DIS
LIN {X 10.1666,Y -5.3035,Z 55,A -33.5727,B 24.8037,C -3.2309,E1 25.1438,E2 -244.2595} C_DIS
LIN {X 10.7138,Y -4.0871,Z 55,A -26.9655,B 24.8013,C -3.2501,E1 25.1509,E2 -250.8759} C_DIS
LIN {X 11.1056,Y -2.8552,Z 55,A -20.53,B 24.7989,C -3.2696,E1 25.1558,E2 -257.3208} C_DIS
LIN {X 11.3609,Y -1.5558,Z 55,A -13.9577,B 24.7964,C -3.2898,E1 25.1589,E2 -263.9024} C_DIS
LIN {X 11.4651,Y -0.1966,Z 55,A -10.6659,B 24.7968,C -3.2869,E1 25.1596,E2 -267.1679} C_DIS
LIN {X 11.4393,Y 0.7941,Z 55,A -2.3668,B 24.792,C -3.3251,E1 25.159,E2 -275.5081} C_DIS
LIN {X 11.2862,Y 2.0267,Z 55,A 3.8307,B 24.7896,C -3.3438,E1 25.1564,E2 -281.7137} C_DIS
LIN {X 10.994,Y 3.2588,Z 55,A 9.1756,B 24.7881,C -3.3559,E1 25.1527,E2 -287.0563} C_DIS
LIN {X 10.7484,Y 3.9948,Z 55,A 13.9633,B 24.7859,C -3.373,E1 25.1482,E2 -291.8578} C_DIS
LIN {X 10.2349,Y 5.1705,Z 55,A 20.4066,B 24.7837,C -3.3906,E1 25.1405,E2 -298.3082} C_DIS
LIN {X 9.5671,Y 6.3214,Z 55,A 27.056,B 24.7815,C -3.4075,E1 25.1307,E2 -304.9638} C_DIS
LIN {X 8.7789,Y 7.3771,Z 55,A 33.5992,B 24.7796,C -3.4224,E1 25.1194,E2 -311.5118} C_DIS
LIN {X 7.9493,Y 8.2643,Z 55,A 39.6784,B 24.7779,C -3.4349,E1 25.1074,E2 -317.595} C_DIS
LIN {X 6.9763,Y 9.1006,Z 55,A 45.8603,B 24.7766,C -3.4452,E1 25.094,E2 -323.7779} C_DIS
LIN {X 5.8172,Y 9.8818,Z 55,A 52.9261,B 24.7752,C -3.456,E1 25.0774,E2 -330.8468} C_DIS
LIN {X 4.6616,Y 10.4764,Z 55,A 59.4179,B 24.7742,C -3.4636,E1 25.061,E2 -337.3396} C_DIS
LIN {X 3.4143,Y 10.9468,Z 55,A 65.0803,B 24.7741,C -3.4646,E1 25.0461,E2 -342.993} C_DIS
LIN {X 2.6035,Y 11.1674,Z 55,A 70.6173,B 24.773,C -3.4728,E1 25.0311,E2 -348.5412} C_DIS
LIN {X 1.1702,Y 11.407,Z 55,A 77.5929,B 24.773,C -3.4732,E1 25.0118,E2 -355.5121} C_DIS
LIN {X -0.1361,Y 11.4661,Z 55,A 84.01,B 24.7731,C -3.4719,E1 24.9939,E2 -361.9251} C_DIS
LIN {X -1.4068,Y 11.3802,Z 55,A 90.3484,B 24.7735,C -3.4687,E1 24.9763,E2 -368.2593} C_DIS
LIN {X -2.6363,Y 11.1597,Z 55,A 96.6106,B 24.7742,C -3.4637,E1 24.9592,E2 -374.5168} C_DIS
LIN {X -3.832,Y 10.8076,Z 55,A 102.9615,B 24.7751,C -3.4569,E1 24.9424,E2 -380.8631} C_DIS
LIN {X -5.003,Y 10.3179,Z 55,A 109.3368,B 24.7763,C -3.4477,E1 24.9262,E2 -387.2321} C_DIS
LIN {X -6.1632,Y 9.6698,Z 55,A 115.4893,B 24.7779,C -3.4352,E1 24.9114,E2 -393.3731} C_DIS
LIN {X -6.8834,Y 9.171,Z 55,A 120.2254,B 24.7789,C -3.4272,E1 24.9007,E2 -398.1067} C_DIS
LIN {X -7.8556,Y 8.3533,Z 55,A 126.995,B 24.7807,C -3.4138,E1 24.8866,E2 -404.8712} C_DIS
LIN {X -8.8132,Y 7.3361,Z 55,A 133.8231,B 24.7829,C -3.3965,E1 24.874,E2 -411.6885} C_DIS
LIN {X -9.5974,Y 6.2755,Z 55,A 140.4734,B 24.7851,C -3.3791,E1 24.8635,E2 -418.3298} C_DIS
LIN {X -10.2607,Y 5.1192,Z 55,A 147.1918,B 24.7875,C -3.3603,E1 24.8546,E2 -425.0389} C_DIS
LIN {X -10.7632,Y 3.9553,Z 55,A 153.5978,B 24.7899,C -3.3417,E1 24.848,E2 -431.436} C_DIS
LIN {X -11.1357,Y 2.7358,Z 55,A 159.8699,B 24.7923,C -3.3222,E1 24.8434,E2 -437.6978} C_DIS
LIN {X -11.3694,Y 1.4913,Z 55,A 166.1637,B 24.7948,C -3.3027,E1 24.8407,E2 -443.9821} C_DIS
LIN {X -11.4641,Y 0.2526,Z 55,A 170.6853,B 24.7973,C -3.2823,E1 24.8398,E2 -448.4821} C_DIS
LIN {X -11.4193,Y -1.0429,Z 55,A -179.1342,B 24.7995,C -3.265,E1 24.8416,E2 -458.6823} C_DIS
LIN {X -10.796,Y -3.8643,Z 55,A -166.1281,B 24.8048,C -3.2212,E1 24.851,E2 -471.6589} C_DIS
LIN {X -10.2539,Y -5.1329,Z 55,A -159.312,B 24.8071,C -3.2024,E1 24.859,E2 -478.467} C_DIS
LIN {X -9.5821,Y -6.2986,Z 55,A -152.5537,B 24.8092,C -3.1855,E1 24.8689,E2 -485.2193} C_DIS
LIN {X -8.9364,Y -7.1855,Z 55,A -146.7699,B 24.8106,C -3.1732,E1 24.8788,E2 -491.0012} C_DIS
LIN {X -7.7846,Y -8.4196,Z 55,A -138.5495,B 24.8128,C -3.1556,E1 24.895,E2 -499.2143} C_DIS
LIN {X -6.744,Y -9.274,Z 55,A -131.8285,B 24.8141,C -3.144,E1 24.9098,E2 -505.9321} C_DIS
LIN {X -5.6712,Y -9.9663,Z 55,A -125.2175,B 24.8151,C -3.1356,E1 24.9256,E2 -512.5433} C_DIS
LIN {X -4.4049,Y -10.5869,Z 55,A -118.3412,B 24.8161,C -3.1276,E1 24.9431,E2 -519.4171} C_DIS
LIN {X -3.141,Y -11.0283,Z 55,A -111.6401,B 24.8166,C -3.1228,E1 24.9609,E2 -526.1187} C_DIS
LIN {X -1.8406,Y -11.3181,Z 55,A -105.1392,B 24.817,C -3.1198,E1 24.9788,E2 -532.6196} C_DIS
LIN {X -0.5937,Y -11.4514,Z 55,A -98.7234,B 24.817,C -3.1202,E1 24.9966,E2 -539.0392} C_DIS
LIN {X -0.5937,Y -11.4514,Z 55,A -98.7234,B 24.817,C -3.1202,E1 24.9966,E2 -539.0392} C_DIS
Enddeposition()
LIN {X 0.0649,Y -10.5035,Z 55,A -97.4738,B 24.8159,C -3.1294,E1 25.0002,E2 -540.3108} C_DIS
Startdeposition()
$VEL.CP = VEL_PRINT
LIN {X -0.9777,Y -10.4627,Z 55,A -104.399,B 24.8164,C -3.1249,E1 24.9808,E2 -533.3726} C_DIS
LIN {X -2.176,Y -10.2805,Z 55,A -111.0159,B 24.8161,C -3.1271,E1 24.9627,E2 -526.754} C_DIS
LIN {X -3.3656,Y -9.9548,Z 55,A -117.8701,B 24.8156,C -3.1314,E1 24.9444,E2 -519.8984} C_DIS
LIN {X -4.9049,Y -9.2933,Z 55,A -127.6898,B 24.8146,C -3.1402,E1 24.9196,E2 -510.0749} C_DIS
LIN {X -6.0085,Y -8.6212,Z 55,A -134.723,B 24.8133,C -3.1511,E1 24.9033,E2 -503.0443} C_DIS
LIN {X -7.1902,Y -7.6635,Z 55,A -142.3491,B 24.8113,C -3.1675,E1 24.8872,E2 -495.4277} C_DIS
LIN {X -7.9217,Y -6.9043,Z 55,A -147.9649,B 24.8098,C -3.18,E1 24.8767,E2 -489.8169} C_DIS
LIN {X -8.5175,Y -6.1546,Z 55,A -153.4029,B 24.8084,C -3.192,E1 24.8676,E2 -484.3817} C_DIS
LIN {X -9.1825,Y -5.1096,Z 55,A -160.2287,B 24.8063,C -3.2092,E1 24.8578,E2 -477.5618} C_DIS
LIN {X -9.7031,Y -4.025,Z 55,A -166.1506,B 24.8041,C -3.2276,E1 24.851,E2 -471.6514} C_DIS
LIN {X -10.0359,Y -3.1145,Z 55,A -172.6763,B 24.8023,C -3.2422,E1 24.8453,E2 -465.1235} C_DIS
LIN {X -10.4015,Y -1.4897,Z 55,A 179.9121,B 24.7989,C -3.2699,E1 24.8412,E2 -457.7346} C_DIS
LIN {X -10.4871,Y -0.6662,Z 55,A 173.4273,B 24.7972,C -3.2834,E1 24.8398,E2 -451.2431} C_DIS
LIN {X -10.4429,Y 1.1709,Z 55,A 164.4752,B 24.7933,C -3.3146,E1 24.8412,E2 -442.3122} C_DIS
LIN {X -10.2638,Y 2.2537,Z 55,A 157.9602,B 24.791,C -3.333,E1 24.8446,E2 -435.8026} C_DIS
LIN {X -9.9226,Y 3.459,Z 55,A 151.1127,B 24.7884,C -3.3535,E1 24.8504,E2 -428.9652} C_DIS
LIN {X -9.4376,Y 4.6212,Z 55,A 144.1578,B 24.7859,C -3.3734,E1 24.8584,E2 -422.0199} C_DIS
LIN {X -8.7984,Y 5.7459,Z 55,A 136.2354,B 24.7834,C -3.3923,E1 24.87,E2 -414.1023} C_DIS
LIN {X -7.7666,Y 7.0786,Z 55,A 128.3756,B 24.7803,C -3.4164,E1 24.8839,E2 -406.2639} C_DIS
LIN {X -7.038,Y 7.7989,Z 55,A 122.9372,B 24.7787,C -3.4293,E1 24.8949,E2 -400.834} C_DIS
LIN {X -6.0198,Y 8.6131,Z 55,A 114.6539,B 24.777,C -3.4421,E1 24.9133,E2 -392.5517} C_DIS
LIN {X -4.9945,Y 9.2456,Z 55,A 108.4171,B 24.7755,C -3.4538,E1 24.9284,E2 -386.3245} C_DIS
LIN {X -3.8475,Y 9.7786,Z 55,A 101.5719,B 24.7742,C -3.4636,E1 24.946,E2 -379.4866} C_DIS
LIN {X -2.6917,Y 10.1576,Z 55,A 94.8872,B 24.7733,C -3.4705,E1 24.9638,E2 -372.8073} C_DIS
LIN {X -1.4436,Y 10.4087,Z 55,A 87.9728,B 24.7726,C -3.4755,E1 24.9829,E2 -365.8982} C_DIS
LIN {X -0.2165,Y 10.5061,Z 55,A 81.2729,B 24.7723,C -3.4779,E1 25.0015,E2 -359.2022} C_DIS
LIN {X 1.6108,Y 10.384,Z 55,A 69.8914,B 24.7731,C -3.4718,E1 25.0331,E2 -347.8139} C_DIS
LIN {X 3.0845,Y 10.0453,Z 55,A 62.9769,B 24.7731,C -3.4718,E1 25.0517,E2 -340.9105} C_DIS
LIN {X 4.392,Y 9.5464,Z 55,A 55.5963,B 24.774,C -3.4652,E1 25.0707,E2 -333.5312} C_DIS
LIN {X 5.2406,Y 9.1082,Z 55,A 50.2527,B 24.775,C -3.4576,E1 25.0838,E2 -328.1853} C_DIS
LIN {X 6.3347,Y 8.3844,Z 55,A 43.046,B 24.7765,C -3.4458,E1 25.1002,E2 -320.9753} C_DIS
LIN {X 7.406,Y 7.455,Z 55,A 34.931,B 24.7788,C -3.4286,E1 25.1168,E2 -312.8525} C_DIS
LIN {X 8.3418,Y 6.3907,Z 55,A 27.6273,B 24.7807,C -3.4134,E1 25.1298,E2 -305.5465} C_DIS
LIN {X 9.055,Y 5.3323,Z 55,A 20.6764,B 24.783,C -3.396,E1 25.1402,E2 -298.5893} C_DIS
LIN {X 9.6661,Y 4.1211,Z 55,A 13.8346,B 24.7851,C -3.3793,E1 25.1483,E2 -291.7447} C_DIS
LIN {X 9.9891,Y 3.2609,Z 55,A 8.171,B 24.7875,C -3.3609,E1 25.1535,E2 -286.0693} C_DIS
LIN {X 10.326,Y 1.9485,Z 55,A 1.1224,B 24.79,C -3.341,E1 25.1578,E2 -279.0145} C_DIS
LIN {X 10.4838,Y 0.7186,Z 55,A -5.6589,B 24.7926,C -3.3201,E1 25.1597,E2 -272.2239} C_DIS
LIN {X 10.5053,Y -0.2527,Z 55,A -11.011,B 24.7947,C -3.3033,E1 25.1595,E2 -266.8638} C_DIS
LIN {X 10.3958,Y -1.5341,Z 55,A -17.9402,B 24.7974,C -3.2821,E1 25.1573,E2 -259.9252} C_DIS
LIN {X 10.1424,Y -2.749,Z 55,A -24.6263,B 24.7999,C -3.2619,E1 25.1529,E2 -253.2298} C_DIS
LIN {X 9.738,Y -3.9491,Z 55,A -31.3924,B 24.8023,C -3.2421,E1 25.1464,E2 -246.4547} C_DIS
LIN {X 9.2019,Y -5.0746,Z 55,A -38.4206,B 24.8048,C -3.2213,E1 25.1374,E2 -239.4142} C_DIS
LIN {X 8.495,Y -6.1856,Z 55,A -45.3226,B 24.807,C -3.2036,E1 25.1265,E2 -232.5045} C_DIS
LIN {X 7.7467,Y -7.1003,Z 55,A -53.1031,B 24.8098,C -3.18,E1 25.1121,E2 -224.7027} C_DIS
LIN {X 6.1537,Y -8.5181,Z 55,A -63.2908,B 24.8119,C -3.163,E1 25.0901,E2 -214.5133} C_DIS
LIN {X 4.863,Y -9.3148,Z 55,A -72.0119,B 24.8139,C -3.1464,E1 25.069,E2 -205.7789} C_DIS
LIN {X 3.4381,Y -9.9293,Z 55,A -80.8432,B 24.8154,C -3.1335,E1 25.0459,E2 -196.9361} C_DIS
LIN {X 2.2699,Y -10.2603,Z 55,A -87.1258,B 24.816,C -3.1286,E1 25.0289,E2 -190.651} C_DIS
LIN {X 0.9058,Y -10.4692,Z 55,A -94.0962,B 24.8162,C -3.1263,E1 25.0096,E2 -183.6804} C_DIS
LIN {X 0.0649,Y -10.5035,Z 55,A -97.4738,B 24.8159,C -3.1294,E1 25.0002,E2 -180.3108} C_DIS
Enddeposition()
LIN {X 0.0649,Y -10.5035,Z 55,A -97.4738,B 24.8159,C -3.1294,E1 25.0002,E2 -180.3108} C_DIS
Startdeposition()
$VEL.CP = VEL_PRINT
LIN {X 0.6074,Y -9.5304,Z 55,A -92.0595,B 24.5259,C -3.084,E1 24.7223,E2 -185.7013} C_DIS
LIN {X 1.7459,Y -9.3886,Z 55,A -85.8773,B 24.5256,C -3.086,E1 24.7393,E2 -191.8825} C_DIS
LIN {X 2.8802,Y -9.1049,Z 55,A -77.1488,B 24.5239,C -3.1007,E1 24.7628,E2 -200.6316} C_DIS
LIN {X 4.1673,Y -8.5924,Z 55,A -68.6495,B 24.5223,C -3.1139,E1 24.7844,E2 -209.1411} C_DIS
LIN {X 5.8026,Y -7.5847,Z 55,A -58.6655,B 24.5206,C -3.128,E1 24.8075,E2 -219.125} C_DIS
LIN {X 6.8561,Y -6.6476,Z 55,A -50.1391,B 24.5183,C -3.1476,E1 24.8249,E2 -227.6632} C_DIS
LIN {X 7.6131,Y -5.7655,Z 55,A -43.4764,B 24.5163,C -3.1636,E1 24.8367,E2 -234.3328} C_DIS
LIN {X 8.222,Y -4.8579,Z 55,A -35.7043,B 24.5133,C -3.1887,E1 24.8482,E2 -242.1253} C_DIS
LIN {X 8.8513,Y -3.5848,Z 55,A -27.9552,B 24.5108,C -3.2088,E1 24.857,E2 -249.88} C_DIS
LIN {X 9.2174,Y -2.4976,Z 55,A -21.0794,B 24.5083,C -3.2296,E1 24.8626,E2 -256.7658} C_DIS
LIN {X 9.4533,Y -1.3536,Z 55,A -14.6131,B 24.506,C -3.2478,E1 24.8657,E2 -263.2374} C_DIS
Enddeposition()
END
